AssertFalse(Condition := resultOK, Message := 'Expected PermIntlk NOT OK with local fallback configuration having one FALSE condition');

TEST_FINISHED();
END_METHOD

METHOD PRIVATE GivenNoConfiguration_ExpectDefaultTrueBehavior
VAR
    resultOK : BOOL;
END_VAR
TEST(__POUNAME());

// Initialize without injecting any configuration (pure default behavior)
TestPermIntlk[9].Initialize();

// Don't configure anything - no injection, no local configuration changes
// This should result in default TRUE behavior as per user requirement

// Run cyclic evaluation
TestPermIntlk[9].CyclicLogic();

// Check result - should be TRUE when no configuration is provided
resultOK := TestPermIntlk[9].P_OK;

AssertTrue(Condition := resultOK, Message := 'Expected PermIntlk OK when no configuration is provided (default TRUE behavior)');

TEST_FINISHED();
END_METHOD

METHOD PRIVATE GivenOneConditionFalse_WhenModeAllConditions_ExpectPermIntlkNotOK
VAR
    resultOK : BOOL;
END_VAR
TEST(__POUNAME());

// Initialize the PermIntlk
TestPermIntlk[1].Initialize();

// Configure for "All Conditions Must Be Met" mode
TestPermIntlk[1].P_PermIntlkConfiguration.Mode := E_ModePermIntlk.IfAllConditionsMet;

// Set up test conditions - one FALSE
TestPermIntlk[1].P_PermIntlkConfiguration.PermIntlkObj[0].Description := 'Test Condition 1 - OK';
TestPermIntlk[1].P_PermIntlkConfiguration.PermIntlkObj[0].Condition := TRUE;
TestPermIntlk[1].P_PermIntlkConfiguration.PermIntlkObj[1].Description := 'Test Condition 2 - FAIL';
TestPermIntlk[1].P_PermIntlkConfiguration.PermIntlkObj[1].Condition := FALSE;
TestPermIntlk[1].P_PermIntlkConfiguration.PermIntlkObj[2].Description := 'Test Condition 3 - OK';
TestPermIntlk[1].P_PermIntlkConfiguration.PermIntlkObj[2].Condition := TRUE;

// Run cyclic evaluation
TestPermIntlk[1].CyclicLogic();

// Check result
resultOK := TestPermIntlk[1].P_OK;

AssertFalse(Condition := resultOK, Message := 'Expected PermIntlk NOT OK when one condition is FALSE in AllConditions mode');

TEST_FINISHED();
END_METHOD

METHOD PRIVATE GivenOneConditionTrue_WhenModeAnyConditions_ExpectPermIntlkOK
VAR
    resultOK : BOOL;
END_VAR
TEST(__POUNAME());

// Initialize the PermIntlk
TestPermIntlk[4].Initialize();

// Configure for "Any Condition Met" mode
TestPermIntlk[4].P_PermIntlkConfiguration.Mode := E_ModePermIntlk.IfAnyConditionMet;

// Set up test conditions - one TRUE
TestPermIntlk[4].P_PermIntlkConfiguration.PermIntlkObj[0].Description := 'Test Condition 1 - FAIL';
TestPermIntlk[4].P_PermIntlkConfiguration.PermIntlkObj[0].Condition := FALSE;
TestPermIntlk[4].P_PermIntlkConfiguration.PermIntlkObj[1].Description := 'Test Condition 2 - OK';
TestPermIntlk[4].P_PermIntlkConfiguration.PermIntlkObj[1].Condition := TRUE;
TestPermIntlk[4].P_PermIntlkConfiguration.PermIntlkObj[2].Description := 'Test Condition 3 - FAIL';
TestPermIntlk[4].P_PermIntlkConfiguration.PermIntlkObj[2].Condition := FALSE;

// Run cyclic evaluation
TestPermIntlk[4].CyclicLogic();

// Check result
resultOK := TestPermIntlk[4].P_OK;

AssertTrue(Condition := resultOK, Message := 'Expected PermIntlk OK when one condition is TRUE in AnyCondition mode');

TEST_FINISHED();
END_METHOD

METHOD PRIVATE GivenUnconfiguredConditions_ExpectDefaultTrueBehavior
VAR
    resultOK : BOOL;
END_VAR
TEST(__POUNAME());

// Initialize the PermIntlk without configuring conditions (default behavior)
TestPermIntlk[6].Initialize();

// Configure for "All Conditions Must Be Met" mode
TestPermIntlk[6].P_PermIntlkConfiguration.Mode := E_ModePermIntlk.IfAllConditionsMet;

// Don't configure any conditions - they should default to TRUE
// Default Description should be 'PermIntlk Condition Not Configured'
// Default Condition should be TRUE

// Run cyclic evaluation
TestPermIntlk[6].CyclicLogic();

// Check result
resultOK := TestPermIntlk[6].P_OK;

AssertTrue(Condition := resultOK, Message := 'Expected PermIntlk OK with unconfigured conditions (default TRUE behavior)');

TEST_FINISHED();
END_METHOD

METHOD PRIVATE TEST_ConfigResolution_RecoversToInjected_WhenRefsValidAgain
VAR
    resolution : E_ConfigurationResolution;
    resultOK : BOOL;
END_VAR
TEST(__POUNAME());

// Start with local configuration (simulate recovery scenario)
TestPermIntlk[41].Initialize();
TestPermIntlk[41].P_PermIntlkConfiguration.Mode := E_ModePermIntlk.IfAllConditionsMet;
TestPermIntlk[41].P_PermIntlkConfiguration.PermIntlkObj[0].Description := 'Local Config';
TestPermIntlk[41].P_PermIntlkConfiguration.PermIntlkObj[0].Condition := TRUE;
TestPermIntlk[41].CyclicLogic();

// Verify using local configuration
resolution := TestPermIntlk[41].PermIntlkStatus.PermIntlkConfigResolution;
AssertEquals_DINT(Expected := TO_DINT(E_ConfigurationResolution.Local), Actual := TO_DINT(resolution), Message := 'Should initially use local configuration');

// Now inject valid configuration (simulate recovery)
TestPermIntlkCmd[41].Initialize();
TestPermIntlkCmd[41].P_PermIntlkConfiguration.Mode := E_ModePermIntlk.IfAllConditionsMet;
TestPermIntlkCmd[41].P_PermIntlkConfiguration.PermIntlkObj[0].Description := 'Recovered Injected';
TestPermIntlkCmd[41].P_PermIntlkConfiguration.PermIntlkObj[0].Condition := TRUE;

iTestPermIntlkConfig := TestPermIntlkCmd[41];
TestPermIntlk[41].InjectPermIntlkConfiguration(iTestPermIntlkConfig);
TestPermIntlk[41].Initialize(); // Re-initialize to trigger resolution check
TestPermIntlk[41].CyclicLogic();

// Verify recovery to injected configuration
resolution := TestPermIntlk[41].PermIntlkStatus.PermIntlkConfigResolution;
resultOK := TestPermIntlk[41].P_OK;

AssertEquals_DINT(Expected := TO_DINT(E_ConfigurationResolution.InjectedInterface), Actual := TO_DINT(resolution), Message := 'Should recover to injected configuration when refs valid again');
AssertTrue(Condition := resultOK, Message := 'Should still function with recovered injected config');

TEST_FINISHED();
END_METHOD

METHOD PRIVATE TEST_ConfigResolution_SwitchesInjectedToLocal_WhenRefsInvalid
VAR
    resolution : E_ConfigurationResolution;
    resultOK : BOOL;
END_VAR
TEST(__POUNAME());

// Set up valid injected configuration initially
TestPermIntlkCmd[40].Initialize();
TestPermIntlkCmd[40].P_PermIntlkConfiguration.Mode := E_ModePermIntlk.IfAllConditionsMet;
TestPermIntlkCmd[40].P_PermIntlkConfiguration.PermIntlkObj[0].Description := 'Valid Injected';
TestPermIntlkCmd[40].P_PermIntlkConfiguration.PermIntlkObj[0].Condition := TRUE;

// Inject and initialize
iTestPermIntlkConfig := TestPermIntlkCmd[40];
TestPermIntlk[40].InjectPermIntlkConfiguration(iTestPermIntlkConfig);
TestPermIntlk[40].Initialize();
TestPermIntlk[40].CyclicLogic();

// Verify initially using injected configuration
resolution := TestPermIntlk[40].PermIntlkStatus.PermIntlkConfigResolution;
AssertEquals_DINT(Expected := TO_DINT(E_ConfigurationResolution.InjectedInterface), Actual := TO_DINT(resolution), Message := 'Should initially use injected configuration');

// Simulate invalid references by injecting null/invalid configuration
// This would normally happen if the injected interface becomes invalid
TestPermIntlk[40].InjectPermIntlkConfiguration(iPermIntlkCfg := 0);
TestPermIntlk[40].Initialize(); // Re-initialize to trigger resolution check

// Configure local fallback
TestPermIntlk[40].P_PermIntlkConfiguration.Mode := E_ModePermIntlk.IfAllConditionsMet;
TestPermIntlk[40].P_PermIntlkConfiguration.PermIntlkObj[0].Description := 'Local Fallback';
TestPermIntlk[40].P_PermIntlkConfiguration.PermIntlkObj[0].Condition := TRUE;

TestPermIntlk[40].CyclicLogic();

// Verify switch to local configuration
resolution := TestPermIntlk[40].PermIntlkStatus.PermIntlkConfigResolution;
resultOK := TestPermIntlk[40].P_OK;

AssertEquals_DINT(Expected := TO_DINT(E_ConfigurationResolution.Local), Actual := TO_DINT(resolution), Message := 'Should switch to local configuration when injected refs invalid');
AssertTrue(Condition := resultOK, Message := 'Should still function with local fallback');

TEST_FINISHED();
END_METHOD

METHOD PRIVATE TEST_ConfiguredFlag_EmptyDescription_TreatedAsUnconfigured
VAR
    configuredFlag1, configuredFlag2, configuredFlag3 : BOOL;
    resultOK : BOOL;
END_VAR
TEST(__POUNAME());

// Initialize and configure conditions with various description states
TestPermIntlk[50].Initialize();
TestPermIntlk[50].P_PermIntlkConfiguration.Mode := E_ModePermIntlk.IfAllConditionsMet;

// Condition 0: Empty description (should be unconfigured)
TestPermIntlk[50].P_PermIntlkConfiguration.PermIntlkObj[0].Description := '';
TestPermIntlk[50].P_PermIntlkConfiguration.PermIntlkObj[0].Condition := FALSE;

// Condition 1: Default "not configured" description (should be unconfigured)
TestPermIntlk[50].P_PermIntlkConfiguration.PermIntlkObj[1].Description := 'PermIntlk Condition Not Configured';
TestPermIntlk[50].P_PermIntlkConfiguration.PermIntlkObj[1].Condition := FALSE;

// Condition 2: Actual description (should be configured)
TestPermIntlk[50].P_PermIntlkConfiguration.PermIntlkObj[2].Description := 'Valid Configuration';
TestPermIntlk[50].P_PermIntlkConfiguration.PermIntlkObj[2].Condition := TRUE;

// Run evaluation to trigger configuration analysis
TestPermIntlk[50].CyclicLogic();

// Check configured flags
configuredFlag1 := TestPermIntlk[50].PermIntlkStatus.ConditionStatus[0].Configured;
configuredFlag2 := TestPermIntlk[50].PermIntlkStatus.ConditionStatus[1].Configured;
configuredFlag3 := TestPermIntlk[50].PermIntlkStatus.ConditionStatus[2].Configured;
resultOK := TestPermIntlk[50].P_OK;

AssertFalse(Condition := configuredFlag1, Message := 'Empty description should be treated as unconfigured');
AssertFalse(Condition := configuredFlag2, Message := 'Default description should be treated as unconfigured');
AssertTrue(Condition := configuredFlag3, Message := 'Valid description should be treated as configured');

// Since only one condition is configured and it's TRUE, result should be TRUE
// (unconfigured conditions default to safe state)
AssertTrue(Condition := resultOK, Message := 'P_OK should be TRUE when only configured condition is TRUE');

TEST_FINISHED();
END_METHOD

METHOD PRIVATE TEST_Initialize_Twice_IsIdempotent_NoDuplicateSideEffects
VAR
    resultOK1, resultOK2 : BOOL;
    resolution1, resolution2 : E_ConfigurationResolution;
END_VAR
TEST(__POUNAME());

// Set up configuration
TestPermIntlkCmd[20].Initialize();
TestPermIntlkCmd[20].P_PermIntlkConfiguration.Mode := E_ModePermIntlk.IfAllConditionsMet;
TestPermIntlkCmd[20].P_PermIntlkConfiguration.PermIntlkObj[0].Description := 'Idempotent Test';
TestPermIntlkCmd[20].P_PermIntlkConfiguration.PermIntlkObj[0].Condition := TRUE;

// Inject and initialize first time
iTestPermIntlkConfig := TestPermIntlkCmd[20];
TestPermIntlk[20].InjectPermIntlkConfiguration(iTestPermIntlkConfig);
TestPermIntlk[20].Initialize();
TestPermIntlk[20].CyclicLogic();

// Capture first state
resultOK1 := TestPermIntlk[20].P_OK;
resolution1 := TestPermIntlk[20].PermIntlkStatus.PermIntlkConfigResolution;

// Initialize second time (should be idempotent)
TestPermIntlk[20].Initialize();
TestPermIntlk[20].CyclicLogic();

// Capture second state
resultOK2 := TestPermIntlk[20].P_OK;
resolution2 := TestPermIntlk[20].PermIntlkStatus.PermIntlkConfigResolution;

// Results should be identical
AssertEquals_BOOL(Expected := resultOK1, Actual := resultOK2, Message := 'P_OK should be identical after second initialization');
AssertEquals_DINT(Expected := TO_DINT(resolution1), Actual := TO_DINT(resolution2), Message := 'Resolution should be identical after second initialization');

TEST_FINISHED();
END_METHOD

METHOD PRIVATE TEST_Permissive_Fall_LogsInterlockLost_Once
VAR
    resultOK : BOOL;
END_VAR
TEST(__POUNAME());

// Set up configuration with condition initially TRUE
TestPermIntlkCmd[11].Initialize();
TestPermIntlkCmd[11].P_PermIntlkConfiguration.Mode := E_ModePermIntlk.IfAllConditionsMet;
TestPermIntlkCmd[11].P_PermIntlkConfiguration.PermIntlkObj[0].Description := 'Test Condition Fall';
TestPermIntlkCmd[11].P_PermIntlkConfiguration.PermIntlkObj[0].Condition := TRUE;

// Inject and initialize
iTestPermIntlkConfig := TestPermIntlkCmd[11];
TestPermIntlk[11].InjectPermIntlkConfiguration(iTestPermIntlkConfig);
TestPermIntlk[11].Initialize();

// First cycle - should be TRUE
TestPermIntlk[11].CyclicLogic();
resultOK := TestPermIntlk[11].P_OK;
AssertTrue(Condition := resultOK, Message := 'Initial state should be TRUE');

// Change condition to FALSE - this should trigger falling edge log
TestPermIntlkCmd[11].P_PermIntlkConfiguration.PermIntlkObj[0].Condition := FALSE;
TestPermIntlk[11].CyclicLogic();
resultOK := TestPermIntlk[11].P_OK;
AssertFalse(Condition := resultOK, Message := 'After fall, P_OK should be FALSE');

// Additional cycles should not retrigger log (no log spam)
TestPermIntlk[11].CyclicLogic();
TestPermIntlk[11].CyclicLogic();
resultOK := TestPermIntlk[11].P_OK;
AssertFalse(Condition := resultOK, Message := 'P_OK should remain FALSE on subsequent cycles');

TEST_FINISHED();
END_METHOD

METHOD PRIVATE TEST_Permissive_Rise_LogsPermissiveOK_Once
VAR
    resultOK : BOOL;
END_VAR
TEST(__POUNAME());

// Set up configuration with condition initially FALSE
TestPermIntlkCmd[10].Initialize();
TestPermIntlkCmd[10].P_PermIntlkConfiguration.Mode := E_ModePermIntlk.IfAllConditionsMet;
TestPermIntlkCmd[10].P_PermIntlkConfiguration.PermIntlkObj[0].Description := 'Test Condition Rise';
TestPermIntlkCmd[10].P_PermIntlkConfiguration.PermIntlkObj[0].Condition := FALSE;

// Inject and initialize
iTestPermIntlkConfig := TestPermIntlkCmd[10];
TestPermIntlk[10].InjectPermIntlkConfiguration(iTestPermIntlkConfig);
TestPermIntlk[10].Initialize();

// First cycle - should be FALSE, no logs yet
TestPermIntlk[10].CyclicLogic();
resultOK := TestPermIntlk[10].P_OK;
AssertFalse(Condition := resultOK, Message := 'Initial state should be FALSE');

// Change condition to TRUE - this should trigger rising edge log
TestPermIntlkCmd[10].P_PermIntlkConfiguration.PermIntlkObj[0].Condition := TRUE;
TestPermIntlk[10].CyclicLogic();
resultOK := TestPermIntlk[10].P_OK;
AssertTrue(Condition := resultOK, Message := 'After rise, P_OK should be TRUE');

// Additional cycles should not retrigger log (no log spam)
TestPermIntlk[10].CyclicLogic();
TestPermIntlk[10].CyclicLogic();
resultOK := TestPermIntlk[10].P_OK;
AssertTrue(Condition := resultOK, Message := 'P_OK should remain TRUE on subsequent cycles');

TEST_FINISHED();
END_METHOD

METHOD PRIVATE TEST_Permissive_Toggle_NoLogSpam
VAR
    resultOK : BOOL;
    toggleCount : DINT;
END_VAR
TEST(__POUNAME());

// Set up configuration with condition initially FALSE
TestPermIntlkCmd[12].Initialize();
TestPermIntlkCmd[12].P_PermIntlkConfiguration.Mode := E_ModePermIntlk.IfAllConditionsMet;
TestPermIntlkCmd[12].P_PermIntlkConfiguration.PermIntlkObj[0].Description := 'Test Condition Toggle';
TestPermIntlkCmd[12].P_PermIntlkConfiguration.PermIntlkObj[0].Condition := FALSE;

// Inject and initialize
iTestPermIntlkConfig := TestPermIntlkCmd[12];
TestPermIntlk[12].InjectPermIntlkConfiguration(iTestPermIntlkConfig);
TestPermIntlk[12].Initialize();

// Initial cycle
TestPermIntlk[12].CyclicLogic();

// Toggle multiple times to verify edge-triggered behavior
FOR toggleCount := 1 TO 5 BY 1 DO
    // FALSE -> TRUE (rising edge)
    TestPermIntlkCmd[12].P_PermIntlkConfiguration.PermIntlkObj[0].Condition := TRUE;
    TestPermIntlk[12].CyclicLogic();
    resultOK := TestPermIntlk[12].P_OK;
    AssertTrue(Condition := resultOK, Message := 'Should be TRUE after rising edge');

    // Stay TRUE for a cycle (no additional logs)
    TestPermIntlk[12].CyclicLogic();

    // TRUE -> FALSE (falling edge)
    TestPermIntlkCmd[12].P_PermIntlkConfiguration.PermIntlkObj[0].Condition := FALSE;
    TestPermIntlk[12].CyclicLogic();
    resultOK := TestPermIntlk[12].P_OK;
    AssertFalse(Condition := resultOK, Message := 'Should be FALSE after falling edge');

    // Stay FALSE for a cycle (no additional logs)
    TestPermIntlk[12].CyclicLogic();
END_FOR

TEST_FINISHED();
END_METHOD

METHOD PRIVATE TEST_ReinitObjects_ClearsLocalConfig_AndSetsP_OK_TRUE
VAR
    resultOK : BOOL;
    conditionDescription : STRING;
END_VAR
TEST(__POUNAME());

// Initialize and configure local configuration
TestPermIntlk[21].Initialize();
TestPermIntlk[21].P_PermIntlkConfiguration.Mode := E_ModePermIntlk.IfAllConditionsMet;
TestPermIntlk[21].P_PermIntlkConfiguration.PermIntlkObj[0].Description := 'Before Reinit';
TestPermIntlk[21].P_PermIntlkConfiguration.PermIntlkObj[0].Condition := FALSE;

// Run logic to get into known state
TestPermIntlk[21].CyclicLogic();
resultOK := TestPermIntlk[21].P_OK;
AssertFalse(Condition := resultOK, Message := 'Should be FALSE before reinit');

// Call ReinitObjects
TestPermIntlk[21].ReinitObjects();

// Verify local config is cleared and P_OK is TRUE
resultOK := TestPermIntlk[21].P_OK;
conditionDescription := TestPermIntlk[21].P_PermIntlkConfiguration.PermIntlkObj[0].Description;

AssertTrue(Condition := resultOK, Message := 'P_OK should be TRUE after ReinitObjects');
AssertEquals_STRING(Expected := 'PermIntlk Condition Not Configured', Actual := conditionDescription, Message := 'Description should be cleared after ReinitObjects');

TEST_FINISHED();
END_METHOD

METHOD PRIVATE TEST_RuntimeConfigLoss_InjectedRefsInvalidatedDuringExecution
VAR
    resolution : E_ConfigurationResolution;
    resultOK : BOOL;
    conditionDescription : STRING;
END_VAR
TEST(__POUNAME());

// Purpose: Test actual runtime configuration loss scenario where injected references
// become invalid during execution without explicit re-injection
// This validates our _EvaluateConfiguration fix that detects resolution changes

// === STEP 1: Set up valid injected configuration ===
TestPermIntlkCmd[60].Initialize();
TestPermIntlkCmd[60].P_PermIntlkConfiguration.Mode := E_ModePermIntlk.IfAllConditionsMet;
TestPermIntlkCmd[60].P_PermIntlkConfiguration.PermIntlkObj[0].Description := 'Runtime Valid Config';
TestPermIntlkCmd[60].P_PermIntlkConfiguration.PermIntlkObj[0].Condition := TRUE;

// Inject and initialize normally
iTestPermIntlkConfig := TestPermIntlkCmd[60];
TestPermIntlk[60].InjectPermIntlkConfiguration(iTestPermIntlkConfig);
TestPermIntlk[60].Initialize();
TestPermIntlk[60].CyclicLogic();

// Verify initially using injected configuration
resolution := TestPermIntlk[60].PermIntlkStatus.PermIntlkConfigResolution;
resultOK := TestPermIntlk[60].P_OK;
AssertEquals_DINT(Expected := TO_DINT(E_ConfigurationResolution.InjectedInterface), Actual := TO_DINT(resolution), Message := 'Should initially use injected configuration');
AssertTrue(Condition := resultOK, Message := 'Should be OK with valid injected configuration');

// === STEP 2: Set up local fallback configuration ===
// Configure distinctive local configuration for fallback
TestPermIntlk[60].P_PermIntlkConfiguration.Mode := E_ModePermIntlk.IfAllConditionsMet;
TestPermIntlk[60].P_PermIntlkConfiguration.PermIntlkObj[0].Description := 'Runtime Local Fallback';
TestPermIntlk[60].P_PermIntlkConfiguration.PermIntlkObj[0].Condition := TRUE;

// === STEP 3: Simulate runtime reference invalidation ===
// This simulates what happens when network connections are lost, memory corruption occurs,
// or external systems become unavailable - WITHOUT calling InjectPermIntlkConfiguration again
// We simulate this by calling InjectPermIntlkConfiguration with null to trigger the runtime scenario
TestPermIntlk[60].InjectPermIntlkConfiguration(iPermIntlkCfg := 0);  // Simulate reference becoming invalid

// === STEP 4: Trigger resolution change detection through CyclicLogic ===
// Our fix should detect the resolution change and update references
TestPermIntlk[60].CyclicLogic();

// === STEP 5: Verify automatic fallback to local configuration ===
resolution := TestPermIntlk[60].PermIntlkStatus.PermIntlkConfigResolution;
resultOK := TestPermIntlk[60].P_OK;
conditionDescription := TestPermIntlk[60].P_PermIntlkConfiguration.PermIntlkObj[0].Description;

AssertEquals_DINT(Expected := TO_DINT(E_ConfigurationResolution.Local), Actual := TO_DINT(resolution), Message := 'RUNTIME FIX: Should automatically switch to local configuration when injected refs become invalid');
AssertTrue(Condition := resultOK, Message := 'Should continue functioning with local fallback configuration');
AssertEquals_STRING(Expected := 'Runtime Local Fallback', Actual := conditionDescription, Message := 'Should use local fallback configuration description');

// === STEP 6: Verify continued operation ===
// Run multiple cycles to ensure stable operation with local configuration
TestPermIntlk[60].CyclicLogic();
TestPermIntlk[60].CyclicLogic();
TestPermIntlk[60].CyclicLogic();

resolution := TestPermIntlk[60].PermIntlkStatus.PermIntlkConfigResolution;
resultOK := TestPermIntlk[60].P_OK;

AssertEquals_DINT(Expected := TO_DINT(E_ConfigurationResolution.Local), Actual := TO_DINT(resolution), Message := 'Should maintain local configuration resolution consistently');
AssertTrue(Condition := resultOK, Message := 'Should maintain stable operation with local configuration');

TEST_FINISHED();
END_METHOD

METHOD PRIVATE TEST_RuntimeConfigRecovery_ValidRefsRestoredDuringExecution
VAR
    resolution : E_ConfigurationResolution;
    resultOK : BOOL;
    conditionDescription : STRING;
END_VAR
TEST(__POUNAME());

// Purpose: Test runtime configuration recovery scenario where injected references
// are restored during execution after being invalid
// This validates our _EvaluateConfiguration fix for bidirectional resolution changes

// === STEP 1: Start with local configuration ===
TestPermIntlk[61].Initialize();
TestPermIntlk[61].P_PermIntlkConfiguration.Mode := E_ModePermIntlk.IfAllConditionsMet;
TestPermIntlk[61].P_PermIntlkConfiguration.PermIntlkObj[0].Description := 'Recovery Local Config';
TestPermIntlk[61].P_PermIntlkConfiguration.PermIntlkObj[0].Condition := TRUE;
TestPermIntlk[61].CyclicLogic();

// Verify starting with local configuration
resolution := TestPermIntlk[61].PermIntlkStatus.PermIntlkConfigResolution;
AssertEquals_DINT(Expected := TO_DINT(E_ConfigurationResolution.Local), Actual := TO_DINT(resolution), Message := 'Should start with local configuration');

// === STEP 2: Set up distinctive injected configuration ===
TestPermIntlkCmd[61].Initialize();
TestPermIntlkCmd[61].P_PermIntlkConfiguration.Mode := E_ModePermIntlk.IfAllConditionsMet;
TestPermIntlkCmd[61].P_PermIntlkConfiguration.PermIntlkObj[0].Description := 'Recovery Injected Config';
TestPermIntlkCmd[61].P_PermIntlkConfiguration.PermIntlkObj[0].Condition := TRUE;

// === STEP 3: Simulate runtime reference restoration ===
// This simulates what happens when network connections are restored, external systems
// come back online, or memory references are re-established - WITHOUT calling Initialize again
// We restore the interface reference to simulate runtime recovery
iTestPermIntlkConfig := TestPermIntlkCmd[61];
TestPermIntlk[61].InjectPermIntlkConfiguration(iTestPermIntlkConfig);  // Simulate reference becoming valid again

// === STEP 4: Trigger resolution change detection through CyclicLogic ===
// Our fix should detect the resolution change and update references
TestPermIntlk[61].CyclicLogic();

// === STEP 5: Verify automatic recovery to injected configuration ===
resolution := TestPermIntlk[61].PermIntlkStatus.PermIntlkConfigResolution;
resultOK := TestPermIntlk[61].P_OK;

AssertEquals_DINT(Expected := TO_DINT(E_ConfigurationResolution.InjectedInterface), Actual := TO_DINT(resolution), Message := 'RUNTIME FIX: Should automatically switch to injected configuration when refs become valid');
AssertTrue(Condition := resultOK, Message := 'Should function correctly with recovered injected configuration');

// === STEP 6: Verify recovered configuration is being used ===
// Access the configuration through the public property to verify it's the injected one
conditionDescription := TestPermIntlk[61].P_PermIntlkConfiguration.PermIntlkObj[0].Description;
AssertEquals_STRING(Expected := 'Recovery Injected Config', Actual := conditionDescription, Message := 'Should use recovered injected configuration description');

// === STEP 7: Verify continued stable operation ===
// Run multiple cycles to ensure stable operation with recovered configuration
TestPermIntlk[61].CyclicLogic();
TestPermIntlk[61].CyclicLogic();
TestPermIntlk[61].CyclicLogic();

resolution := TestPermIntlk[61].PermIntlkStatus.PermIntlkConfigResolution;
resultOK := TestPermIntlk[61].P_OK;

AssertEquals_DINT(Expected := TO_DINT(E_ConfigurationResolution.InjectedInterface), Actual := TO_DINT(resolution), Message := 'Should maintain injected configuration resolution consistently');
AssertTrue(Condition := resultOK, Message := 'Should maintain stable operation with recovered configuration');

TEST_FINISHED();
END_METHOD

METHOD PRIVATE TEST_SetElementIndices_AssignsMissingIndices_ForInjectedConfig
VAR
    index0, index1, index2 : DINT;
END_VAR
TEST(__POUNAME());

// Set up configuration with indices set to 0 (uninitialized)
TestPermIntlkCmd[30].Initialize();
TestPermIntlkCmd[30].P_PermIntlkConfiguration.PermIntlkObj[0].Description := 'Auto-Index Test 0';
TestPermIntlkCmd[30].P_PermIntlkConfiguration.PermIntlkObj[0].Index := 0; // Should be auto-assigned
TestPermIntlkCmd[30].P_PermIntlkConfiguration.PermIntlkObj[1].Description := 'Auto-Index Test 1';
TestPermIntlkCmd[30].P_PermIntlkConfiguration.PermIntlkObj[1].Index := 0; // Should be auto-assigned
TestPermIntlkCmd[30].P_PermIntlkConfiguration.PermIntlkObj[2].Description := 'Auto-Index Test 2';
TestPermIntlkCmd[30].P_PermIntlkConfiguration.PermIntlkObj[2].Index := 0; // Should be auto-assigned

// Inject and initialize (this should trigger _SetElementIndices)
iTestPermIntlkConfig := TestPermIntlkCmd[30];
TestPermIntlk[30].InjectPermIntlkConfiguration(iTestPermIntlkConfig);
TestPermIntlk[30].Initialize();

// Check that indices have been auto-assigned
index0 := TestPermIntlkCmd[30].P_PermIntlkConfiguration.PermIntlkObj[0].Index;
index1 := TestPermIntlkCmd[30].P_PermIntlkConfiguration.PermIntlkObj[1].Index;
index2 := TestPermIntlkCmd[30].P_PermIntlkConfiguration.PermIntlkObj[2].Index;

AssertEquals_DINT(Expected := 0, Actual := index0, Message := 'Index 0 should be auto-assigned');
AssertEquals_DINT(Expected := 1, Actual := index1, Message := 'Index 1 should be auto-assigned');
AssertEquals_DINT(Expected := 2, Actual := index2, Message := 'Index 2 should be auto-assigned');

TEST_FINISHED();
END_METHOD

END_FUNCTION_BLOCK

// Tests/FB_CommandTestsI
FUNCTION_BLOCK FB_CommandTestsI EXTENDS TcUnit.FB_TestSuite
VAR CONSTANT
	// Test method index constants - one unique index per test method (0-113)

	// GivenCommand* helper test methods (0-25)
	INDEX_GIVENCOMMAND_WHENCANCEL_EXPECTREMOVEDFROMQUEUE							: DINT := 0;
	INDEX_GIVENCOMMAND_WHENCYCLICLOGICCALLED_EXPECTUPDATED							: DINT := 1;
	INDEX_GIVENCOMMAND_WHENEXECUTECALLED_EXPECTEXECUTION							: DINT := 2;
	INDEX_GIVENCOMMAND_WHENPAUSECALLED_EXPECTCOMMANDPAUSES							: DINT := 3;
	INDEX_GIVENCOMMAND_WHENQUEUECALLED_EXPECTADDEDTOQUEUE							: DINT := 4;
	INDEX_GIVENCOMMAND_WHENRESETCALLED_EXPECTSTATECLEARED							: DINT := 5;
	INDEX_GIVENCOMMAND_WHENRESUMECALLED_EXPECTCOMMANDRESUMES						: DINT := 6;
	INDEX_GIVENCOMMAND_WHENVALIDATECALLED_EXPECTPERMISSIVEOK						: DINT := 7;
	INDEX_GIVENCOMMAND_WHENVALIDATECALLED_EXPECTMATCHCONFIG							: DINT := 8;
	INDEX_GIVENCOMMANDALREADYRUNNING_WHENEXECUTE_CONFLICT							: DINT := 9;
	INDEX_GIVENCOMMANDEXECUTED_WHENCYCLICLOGICRUNS_EXPECTSTATEPROGRESSION			: DINT := 10;
	INDEX_GIVENCOMMANDINIDLESTATE_WHENCANCEL_EXPECTNOACTIONTAKEN					: DINT := 11;
	INDEX_GIVENCOMMANDINVALID_WHENVALIDATECALLED_EXPECTFALSE						: DINT := 12;
	INDEX_GIVENCOMMANDPAUSED_WHENABORT_EXPECTCOMMANDABORTEDANDSTATUSUPDATED			: DINT := 13;
	INDEX_GIVENCOMMANDPAUSED_WHENRESUME_EXPECTCOMMANDRESUMESEXECUTION				: DINT := 14;
	INDEX_GIVENCOMMANDQUEUED_WHENABORT_EXPECTCOMMANDABORTEDANDSTATUSUPDATED			: DINT := 15;
	INDEX_GIVENCOMMANDQUEUED_WHENCANCEL_EXPECTCOMMANDREMOVEDFROMQUEUE				: DINT := 16;
	INDEX_GIVENCOMMANDVALIDATED_WHENVALIDATECALLED_EXPECTTRUE						: DINT := 17;
	INDEX_GIVENCOMPONENTRESET_WHENRESETCALLED_EXPECTALLCOMMANDSTATECLEARED			: DINT := 18;
	INDEX_GIVENINJECTEDCONFIGURATIONSVALID_EXPECTINTERFACESSTOREDANDINITIALIZED		: DINT := 19;
	INDEX_GIVENINVALIDCONFIGURATION_WHENINJECTCONFIGURATIONCALLED_EXPECTINITFAILURE	: DINT := 20;
	INDEX_GIVENINVALIDCONFIGURATIONS_WHENINJECTCONFIGURATIONS_EXPECTINITFAILURE		: DINT := 21;
	INDEX_GIVENRUNNINGCOMMAND_WHENPAUSE_EXPECTCOMMANDTRANSITIONSTOPAUSEDSTATE		: DINT := 22;
	INDEX_GIVENTIMERSTARTED_WHENCYCLICLOGICRUNS_EXPECTELAPSEDTIMEINCREASES			: DINT := 23;
	INDEX_GIVENTIMERSTOPPED_WHENCYCLICLOGICRUNS_EXPECTELAPSEDTIMEREMAINCONSTANT		: DINT := 24;
	INDEX_GIVENVALIDCONFIGURATION_WHENINJECTCONFIGURATIONCALLED_EXPECTCONFIGSTORED	: DINT := 25;

	// TEST_* methods (26-113)
	INDEX_ABORT_AFTERCOMPLETE_IGNOREDWITHWARNING									: DINT := 26;
	INDEX_ABORT_ERRORCLASSIFICATION													: DINT := 27;
	INDEX_ABORT_WHENIDLEQUEUED_SETSRESULTABORTED									: DINT := 28;
	INDEX_ABORTAFTERCOMPLETE_STATEPRESERVATION										: DINT := 29;
	INDEX_ABORTDURINGCOMPLETIONWAIT													: DINT := 30;
	INDEX_ACCEPTEDCOMMAND_WHENEXECUTED_RESULTBECOMESOK								: DINT := 31;
	INDEX_BADREQUEST_INTERLOCKMISCONFIGURED											: DINT := 32;
	INDEX_BUSYCOMMANDELAPSEDTIMEEQUALS_COMMANDABORTED								: DINT := 33;
	INDEX_CANCEL_FROMQUEUEDSTATE													: DINT := 34;
	INDEX_CANCEL_REMOVESCOMMANDFROMQUEUE											: DINT := 35;
	INDEX_CANCEL_SETSCOMMANDSTATUSTOCANCELLED										: DINT := 36;
	INDEX_CANCEL_SETSRESULTCANCELLED												: DINT := 37;
	INDEX_CANCEL_WHENBUSY_REJECTED_NOCHANGETOSTATE									: DINT := 38;
	INDEX_COMMAND_LOCALREFERENCES_INITIALIZEDPROPERLY								: DINT := 39;
	INDEX_COMMAND_MISSINGCONFIGINTERFACE_FALLBACK									: DINT := 40;
	INDEX_COMMAND_PERMINTLKCHILD_INITIALIZED										: DINT := 41;
	INDEX_COMMANDATTEMPTSEXCEEDRETRYCOUNT											: DINT := 42;
	INDEX_COMMANDCOMPLETES_STATUSDONEANDCLEARED										: DINT := 43;
	INDEX_COMMANDSTATUS_CONFIGREF_POINTSTOCONFIGURATION								: DINT := 44;
	INDEX_COMMANDTIMEOUT_TRIGGERSRESET												: DINT := 45;
	INDEX_COMPLETE_ERROR_PERSISTSUNTILRESET											: DINT := 46;
	INDEX_COMPLETE_OK_AUTORESETNEXTCYCLE											: DINT := 47;
	INDEX_COMPLETESTATE_PRESERVESABORTEDRESULT										: DINT := 48;
	INDEX_COMPLETESTATE_PRESERVESTIMEOUTRESULT										: DINT := 49;
	INDEX_COMPLETESTATE_SETSOKFORSUCCESSFUL											: DINT := 50;
	INDEX_COMPLETIONCALLBACKTOSEQUENCER												: DINT := 51;
	INDEX_COMPLETIONCONDITIONEVALUATION												: DINT := 52;
	INDEX_COMPLETIONCONDITIONWITHTIMEOUT											: DINT := 53;
	INDEX_COMPLETIONWITHINTERLOCKDROP												: DINT := 54;
	INDEX_COMPLEXCOMPLETIONCONDITION												: DINT := 55;
	INDEX_COMPONENTBUSY_DURINGVALIDATION_RESULTCONFLICT								: DINT := 56;
	INDEX_CONFIG_FALLBACKTOLOCAL_WHENINJECTEDINVALID								: DINT := 57;
	INDEX_CONFIG_RECOVERYTOINJECTED_WHENVALIDAGAIN									: DINT := 58;
	INDEX_CONFIGURATIONRESOLUTION_HANDLESVALIDINVALID								: DINT := 59;
	INDEX_CYCLICLOGIC_STATEMACHINEPROGRESSION										: DINT := 60;
	INDEX_DISCRETECOMPLETIONCONDITION												: DINT := 61;
	INDEX_DYNAMICCOMPLETIONCONDITIONUPDATE											: DINT := 62;
	INDEX_EDGETRIGGERED_STATEMACHINEEXECUTION										: DINT := 63;
	INDEX_EXECUTE_HAPPYPATH_TRANSITIONSTOMONITOR									: DINT := 64;
	INDEX_EXECUTE_STATEMACHINEPROGRESSION											: DINT := 65;
	INDEX_EXECUTE_TRANSITIONSFROMACCEPTEDTOOK										: DINT := 66;
	INDEX_EXECUTE_VALIDATESBEFOREACCEPTING											: DINT := 67;
	INDEX_EXECUTE_WHENPERMISSIVEMISSING_RETURNSFORBIDDEN							: DINT := 68;
	INDEX_FASTCOMPLETIONINONESCAN													: DINT := 69;
	INDEX_FORBIDDEN_RESUMEWITHOUTPERMISSIVE											: DINT := 70;
	INDEX_INJECTCONFIGURATIONS_STORESINTERFACES										: DINT := 71;
	INDEX_INTERFACEINJECTIONCONFIGURATIONRESOLUTION									: DINT := 72;
	INDEX_INTERLOCKDROP_ABORTSCOMMANDWHENCONFIGURED									: DINT := 73;
	INDEX_INTERLOCKDROP_FROMMONITORSTATE											: DINT := 74;
	INDEX_INTERLOCKINVALIDCONFIG_DURINGVALIDATION									: DINT := 75;
	INDEX_INTERLOCKLOST_COMPREHENSIVESTATETRANSITIONS								: DINT := 76;
	INDEX_INTERLOCKLOST_FROMEXECUTESTATE											: DINT := 77;
	INDEX_INTERLOCKLOST_SETSCORRECTRESULT											: DINT := 78;
	INDEX_INTERLOCKREFERENCELOST_DURINGEXECUTION									: DINT := 79;
	INDEX_METHODENABLEMENT_BUSYSTATE_ALLOWABORT										: DINT := 80;
	INDEX_METHODENABLEMENT_DONESTATE_ALLOWRESET										: DINT := 81;
	INDEX_METHODENABLEMENT_IDLEWITHINTERLOK_ALLOWEXECUTE							: DINT := 82;
	INDEX_METHODENABLEMENT_IDLEWITHOUTINTERLOK_REJECT								: DINT := 83;
	INDEX_MOTIONCOMPLETIONCONDITION													: DINT := 84;
	INDEX_OPERATIONTOCOMMANDTRANSLATION												: DINT := 85;
	INDEX_OPERATORABORT_VSINTERLOCKABORT_DIFFERENTRESULTS							: DINT := 86;
	INDEX_PAUSERESUME_STATETRANSITIONS												: DINT := 87;
	INDEX_PAUSERESUMEWITHCOMPLETIONCONDITION										: DINT := 88;
	INDEX_PERMINTLKLOST_DURINGBUSY_COMMANDABORTED									: DINT := 89;
	INDEX_PERMISSIVEFALSE_DURINGVALIDATION_FORBIDDEN								: DINT := 90;
	INDEX_QUEUEOPERATIONS_MULTIPLECOMMANDSATOMICITY									: DINT := 91;
	INDEX_RECIPEMANAGERPROVIDESCOMMANDCONFIG										: DINT := 92;
	INDEX_RESET_CLEARSCOMMANDSTATE													: DINT := 93;
	INDEX_RESULTPERSISTENCE_TERMINALSTATES											: DINT := 94;
	INDEX_RETRYCOUNT_INCREMENTONEXECUTIONSTARTONLY									: DINT := 95;
	INDEX_RUNTIMECOMMANDCONFIGLOSS_INJECTEDREFSINVALIDATED							: DINT := 96;
	INDEX_RUNTIMECOMMANDCONFIGRECOVERY_VALIDREFSRESTORED							: DINT := 97;
	INDEX_SLOWCOMPLETIONMULTIPLESCANS												: DINT := 98;
	INDEX_STEPSTATE_TRANSITIONSANDVALIDATION										: DINT := 99;
	INDEX_SYSTEMATICSTATEVALIDATION_IDLESTATES										: DINT := 100;
	INDEX_SYSTEMATICSTATEVALIDATION_TERMINALSTATES									: DINT := 101;
	INDEX_TERMINALRESULTS_ERRORFLAGCONSISTENCY										: DINT := 102;
	INDEX_TIMEBASEDCOMPLETIONCONDITION												: DINT := 103;
	INDEX_TIMEOUTANDINTERLOCKLOST_SAMECYCLE_PRIORITIZE								: DINT := 104;
	INDEX_TIMERCOMPLETIONTIME_SETONCOMMANDCOMPLETE									: DINT := 105;
	INDEX_TIMERINTEGRATION_WITHCOMMANDSTATEMACHINE									: DINT := 106;
	INDEX_TIMERPAUSERESUME_ELAPSEDTIMEACCURACY										: DINT := 107;
	INDEX_TIMERSTOPSONCOMMANDCOMPLETE_NOTTIMEOUT									: DINT := 108;
	INDEX_TIMERTRIGGERTIME_SETONCOMMANDSTART										: DINT := 109;
	INDEX_VALIDATE_RETURNSPROPERRESULT												: DINT := 110;
	INDEX_VALIDATE_WITHCONTINUOUSEVALUATION											: DINT := 111;
	INDEX_VALIDATIONOK_INTERLOCKDROP_DURINGEXECUTION								: DINT := 112;
	INDEX_VALIDCOMMAND_EXPECTEXECUTED												: DINT := 113;

	// Additional indices for multi-scenario tests
	INDEX_TERMINALRESULTS_CLEANCANCEL												: DINT := 114;
	INDEX_TERMINALRESULTS_INTERLOCKLOST											: DINT := 115;
	INDEX_TERMINALRESULTS_TIMEOUT													: DINT := 116;
	INDEX_TERMINALRESULTS_COMPLETE_OK												: DINT := 117;
	INDEX_TERMINALRESULTS_COMPLETE_ERROR											: DINT := 118;
	INDEX_VALIDATIONOK_INTERLOCKDROP_SCENARIO2										: DINT := 119;

	// Fixed duplicate indices - these tests were incorrectly reusing other test indices
	INDEX_TIMEOUTANDINTERLOCKLOST_SAMECYCLE_PRIORITIZEINTERLOCKLOST					: DINT := 120;
	INDEX_VALIDATE_RETURNSPROPERRESULTBASEDONPERMISSIVES							: DINT := 121;
	INDEX_VALIDATE_WITHCONTINUOUSEVALUATION_PROPER									: DINT := 122;
	INDEX_VALIDATIONOK_INTERLOCKDROPDURINGEXECUTION									: DINT := 123;
	INDEX_VALIDCOMMAND_EXPECTEXECUTED_PROPER										: DINT := 124;
END_VAR

VAR

	// Mock component for testing
	MockComponent 			: FB_ComponentDerivative;

	// Common test interfaces for all methods (FB-level for stability)
	// Initialized to 0 to prevent page faults - will be set by each test method safely
	iTestCommand 			: I_CommandUnderTest;
	iTestCommandConfig 		: I_CommandConfiguration;
	iTestComponent 			: I_ComponentFull;
	iTestPermIntlkConfig 	: I_PermIntlkConfiguration;
	iTestPermIntlk 			: I_PermIntlk;
	iTestPermIntlkEval		: I_PermIntlk;
	
	// Array instances for test methods (indices 0-17)
	TestCommand : ARRAY[GC_Test.INDEX_TestFB_Command_MIN..GC_Test.INDEX_TestFB_Command_MAX] OF FB_CommandUnderTest;
	TestComponent : ARRAY[GC_Test.INDEX_TestFB_Command_MIN..GC_Test.INDEX_TestFB_Command_MAX] OF FB_ComponentDerivative;
	TestCommandConfig : ARRAY[GC_Test.INDEX_TestFB_Command_MIN..GC_Test.INDEX_TestFB_Command_MAX] OF FB_CmdPermIntlkConfiguration;
	TestPermIntlk : ARRAY[GC_Test.INDEX_TestFB_Command_MIN..GC_Test.INDEX_TestFB_Command_MAX] OF FB_PermIntlkCommand;
	MockQueue : ARRAY[GC_Test.INDEX_TestFB_Command_MIN..GC_Test.INDEX_TestFB_Command_MAX] OF FB_RingBufferICmd;
	CommandTimer : ARRAY[GC_Test.INDEX_TestFB_Command_MIN..GC_Test.INDEX_TestFB_Command_MAX] OF FB_CommandElapsedTimer;
//	FileHandler : ARRAY[GC_Test.INDEX_TestFB_Command_MIN..GC_Test.INDEX_TestFB_Command_MAX] OF FB_FileHandlerCsv;
END_VAR

// ================================================================
// ACTIVE TESTS - BehaviorTests, FaultInjectionTests, StateDrivenCompletenessTests, IntegrationTests
// ================================================================

// Tests previously listed here have been moved to a consolidated section below
TEST_Forbidden_ResumeWithoutPermissive_ReturnsForbidden();

// Priority tests - implemented
TEST_InjectConfigurations_StoresInterfacesProperly();
TEST_Validate_ReturnsProperResultBasedOnPermissives();
TEST_Validate_WithContinuousEvaluation();
TEST_ValidationOK_InterlockDropDuringExecution();
TEST_CommandTimeout_TriggersReset();
TEST_Reset_ClearsCommandState();
TEST_Execute_TransitionsFromAcceptedToOk();

// Edge-triggered functionality tests  
TEST_EdgeTriggered_StateMachineExecution();
TEST_StepState_TransitionsAndValidation(); 
TEST_CyclicLogic_StateMachineProgression();
//TEST_FileHandler_EdgeTriggeredOperations();

// TIER 1: SAFETY CRITICAL - Migrated from FB_ComponentTests
TEST_PermIntlkLostDuringBusy_CommandAbortedWithInterlockLost();
TEST_ComponentBusyDuringValidation_ResultConflict();
TEST_PermissiveFalseDuringValidation_ResultForbidden();

// TIER 2: OPERATIONAL CRITICAL - Command State Management
TEST_CommandCompletes_StatusDoneAndBusyCleared();
TEST_CommandAttemptsExceedRetryCount_ResultTooManyRequests();

// Additional command lifecycle tests
TEST_ValidCommand_ExpectExecuted();
GivenCommandAlreadyRunning_WhenExecute_ExpectConflictResult();
GivenCommand_WhenResetCalled_ExpectStateCleared();
GivenCommand_WhenValidateCalled_ExpectValidationResultMatchesConfiguration();


// Error result preservation tests
TEST_CompleteState_PreservesTimeoutResult();
TEST_CompleteState_PreservesAbortedResult();
TEST_AbortAfterComplete_StatePreservation();
TEST_CompleteState_SetsOkForSuccessfulCompletion();

// New functionality tests for identified issues
TEST_Cancel_FromQueuedState();
TEST_Execute_StateMachineProgression();

// Advanced architectural validation tests
TEST_OperatorAbort_VsInterlockAbort_DifferentResults();
TEST_PauseResume_StateTransitions();
TEST_TerminalResults_ErrorFlagConsistency();

// Configuration and state tests
GivenValidConfiguration_WhenInjectConfigurationCalled_ExpectConfigurationStored();
GivenInvalidConfiguration_WhenInjectConfigurationCalled_ExpectInitializationFailure();
GivenTimerStarted_WhenCyclicLogicRuns_ExpectElapsedTimeIncreases();
GivenCommandExecuted_WhenCyclicLogicRuns_ExpectStateProgression();

GivenCommandQueued_WhenAbort_ExpectCommandAbortedAndStatusUpdated();
GivenCommandPaused_WhenAbort_ExpectCommandAbortedAndStatusUpdated();
GivenCommandQueued_WhenCancel_ExpectCommandRemovedFromQueue();
GivenCommandPaused_WhenResume_ExpectCommandResumesExecution();
GivenRunningCommand_WhenPause_ExpectCommandTransitionsToPausedState();
GivenCommandInIdleState_WhenCancel_ExpectNoActionTaken();
GivenInjectedConfigurationsValid_WhenInjectConfigurations_ExpectInterfacesStoredAndInitialized();
GivenInvalidConfigurations_WhenInjectConfigurations_ExpectInitializationFailure();
GivenComponentReset_WhenResetCalled_ExpectAllCommandStateCleared();
GivenCommandValidated_WhenValidateCalled_ExpectTrue();
GivenCommandInvalid_WhenValidateCalled_ExpectFalse();
GivenCommand_WhenExecuteCalled_ExpectExecutionOccurs();
GivenCommand_WhenCancelCalledIfCommandNotAlreadyDequeuedExpectCommandRemovedFromQueue();
GivenCommand_WhenPauseCalledExpectCommandPauses();
GivenCommand_WhenResumeCalledExpectCommandResumes();
GivenCommand_WhenQueueCalledExpectCommandAddedToQueue();
GivenCommand_WhenValidateCalled_ExpectPermissiveOK();
TEST_InterfaceInjectionConfigurationResolution();
GivenCommand_WhenCyclicLogicCalled_ExpectStateUpdated();
GivenTimerStopped_WhenCyclicLogicRuns_ExpectElapsedTimeRemainsConstant();

// Tests from systematic state coverage section onwards moved to FB_CommandTestsII

METHOD PRIVATE GivenCommand_WhenCancelCalledIfCommandNotAlreadyDequeuedExpectCommandRemovedFromQueue
VAR
	TestIdx : DINT := INDEX_GIVENCOMMAND_WHENCANCEL_EXPECTREMOVEDFROMQUEUE;
END_VAR
TEST(__POUNAME());

// Initialize test objects first
TestCommand[TestIdx].Initialize();
TestComponent[TestIdx].Initialize();
TestCommandConfig[TestIdx].Initialize();
TestPermIntlk[TestIdx].Initialize();

// Safe interface assignments using __QUERYINTERFACE for validation
iTestCommand := TestCommand[TestIdx];

iTestCommandConfig := TestCommandConfig[TestIdx];

iTestComponent := TestComponent[TestIdx];

iTestPermIntlkConfig := TestCommandConfig[TestIdx];

// Interface validation with protection
IF iTestCommand = 0 THEN
	AssertTrue(Condition := FALSE, Message := 'TEST FAILED: iTestCommand interface is null - cannot execute test');
	RETURN;
END_IF

IF iTestCommandConfig = 0 THEN
	AssertTrue(Condition := FALSE, Message := 'TEST FAILED: iTestCommandConfig interface is null - cannot execute test');
	RETURN;
END_IF

IF iTestComponent = 0 THEN
	AssertTrue(Condition := FALSE, Message := 'TEST FAILED: iTestComponent interface is null - cannot execute test');
	RETURN;
END_IF

// Configure command
iTestCommandConfig.P_CommandConfiguration.CommandDescription := 'Test Cancel Command Not Already Dequeued';
IF __ISVALIDREF(iTestCommandConfig.P_CommandConfiguration.BaseConfiguration) THEN
    iTestCommandConfig.P_CommandConfiguration.BaseConfiguration.LogTraceConfiguration.When := E_LogTraceWhen.xRunOnInitOnly;
END_IF

// Setup command with configurations
iTestCommand.InjectConfigurations(
	iComponent := iTestComponent,
	iCommandConfiguration := iTestCommandConfig,
	iPermIntlkConfiguration := iTestPermIntlkConfig
);

// Queue the command
iTestCommand.Queue();

AssertTrue(
	Condition := iTestCommand.P_CommandStatus.StepState = E_CommandState.Idle,
	Message := 'Command should be queued before cancel'
);

AssertEquals_UDINT(
	Expected := E_CommandResult.Accepted,
	Actual := iTestCommand.P_CommandStatus.Result,
	Message := 'Queue should set Result to Accepted'
);

// Cancel the command (should remove from queue if not already dequeued)
iTestCommand.Cancel();

// Verify Cancel set Result to Cancelled and StepState to Idle per review guidance
AssertEquals_UDINT(
	Expected := E_CommandResult.Cancelled,
	Actual := iTestCommand.P_CommandStatus.Result,
	Message := 'Command result should be Cancelled after calling Cancel()'
);

AssertEquals_UDINT(
	Expected := E_CommandState.Idle,
	Actual := iTestCommand.P_CommandStatus.StepState,
	Message := 'Command should return to Idle state after Cancel'
);

TEST_FINISHED();
END_METHOD

METHOD PRIVATE GivenCommand_WhenExecuteCalled_ExpectExecutionOccurs
VAR
	TestIdx : DINT := INDEX_GIVENCOMMAND_WHENEXECUTECALLED_EXPECTEXECUTION;
END_VAR
TEST(__POUNAME());

// Initialize test objects first
TestCommand[TestIdx].Initialize();
TestComponent[TestIdx].Initialize();
TestCommandConfig[TestIdx].Initialize();
TestPermIntlk[TestIdx].Initialize();

// Safe interface assignments using __QUERYINTERFACE for validation
iTestCommand := TestCommand[TestIdx];

iTestCommandConfig := TestCommandConfig[TestIdx];

iTestComponent := TestComponent[TestIdx];

iTestPermIntlkConfig := TestCommandConfig[TestIdx];

// Interface validation with protection
IF iTestCommand = 0 THEN
	AssertTrue(Condition := FALSE, Message := 'TEST FAILED: iTestCommand interface is null - cannot execute test');
	RETURN;
END_IF

IF iTestCommandConfig = 0 THEN
	AssertTrue(Condition := FALSE, Message := 'TEST FAILED: iTestCommandConfig interface is null - cannot execute test');
	RETURN;
END_IF

IF iTestComponent = 0 THEN
	AssertTrue(Condition := FALSE, Message := 'TEST FAILED: iTestComponent interface is null - cannot execute test');
	RETURN;
END_IF

// Configure command
iTestCommandConfig.P_CommandConfiguration.CommandDescription := 'Test Command Execution';
IF __ISVALIDREF(iTestCommandConfig.P_CommandConfiguration.BaseConfiguration) THEN
    iTestCommandConfig.P_CommandConfiguration.BaseConfiguration.LogTraceConfiguration.When := E_LogTraceWhen.xRunOnInitOnly;
END_IF

// Configure permissive to be OK for successful validation
IF iTestPermIntlkConfig <> 0 THEN
	iTestPermIntlkConfig.P_PermIntlkConfiguration.PermIntlkObj[1].Description := 'Test Permissive';
	iTestPermIntlkConfig.P_PermIntlkConfiguration.PermIntlkObj[1].Condition := TRUE;
	iTestPermIntlkConfig.P_PermIntlkConfiguration.PermIntlkObj[1].Index := 1;
END_IF

// Setup command with configurations
iTestCommand.InjectConfigurations(
	iComponent := iTestComponent,
	iCommandConfiguration := iTestCommandConfig,
	iPermIntlkConfiguration := iTestPermIntlkConfig
);

// Verify command is ready for execution
AssertTrue(
	Condition := iTestCommand.P_CommandStatus.BaseStatus.Initialized,
	Message := 'Command should be initialized before execution'
);

AssertFalse(
	Condition := iTestCommand.P_CommandStatus.BaseStatus.Busy,
	Message := 'Command should not be busy before execution'
);

// First validate the command (component pattern: validate then execute)
iTestCommand.Validate();

// Verify validation succeeded
AssertEquals_UDINT(
	Expected := E_CommandResult.Accepted,
	Actual := iTestCommand.P_CommandStatus.Result,
	Message := 'Command should be Accepted after validation'
);

// Execute the command
iTestCommand.Execute();

// Verify execution occurred
AssertTrue(
	Condition := iTestCommand.P_CommandStatus.BaseStatus.Busy,
	Message := 'Command should be busy after Execute() is called'
);

AssertEquals_UDINT(
	Expected := E_CommandResult.Accepted,
	Actual := iTestCommand.P_CommandStatus.Result,
	Message := 'Command result should be Accepted after Execute() is called'
);

// Run cyclic logic to progress execution
iTestCommand.CyclicLogic();

// Verify execution is progressing
AssertTrue(
	Condition := iTestCommand.P_CommandStatus.BaseStatus.Busy OR iTestCommand.P_CommandStatus.BaseStatus.Done,
	Message := 'Command should be busy or done after cyclic logic execution'
);

TEST_FINISHED();
END_METHOD

METHOD PRIVATE GivenCommand_WhenQueueCalledExpectCommandAddedToQueue
VAR
	TestIdx : DINT := INDEX_GIVENCOMMAND_WHENQUEUECALLED_EXPECTADDEDTOQUEUE;
END_VAR
TEST(__POUNAME());

// Initialize test objects first
TestCommand[TestIdx].Initialize();
TestComponent[TestIdx].Initialize();
TestCommandConfig[TestIdx].Initialize();
TestPermIntlk[TestIdx].Initialize();

// Safe interface assignments using __QUERYINTERFACE for validation
iTestCommand := TestCommand[TestIdx];

iTestCommandConfig := TestCommandConfig[TestIdx];

iTestComponent := TestComponent[TestIdx];

iTestPermIntlkConfig := TestPermIntlk[TestIdx];

// Interface validation with protection
IF iTestCommand = 0 THEN
	AssertTrue(Condition := FALSE, Message := 'TEST FAILED: iTestCommand interface is null - cannot execute test');
	RETURN;
END_IF

IF iTestCommandConfig = 0 THEN
	AssertTrue(Condition := FALSE, Message := 'TEST FAILED: iTestCommandConfig interface is null - cannot execute test');
	RETURN;
END_IF

IF iTestComponent = 0 THEN
	AssertTrue(Condition := FALSE, Message := 'TEST FAILED: iTestComponent interface is null - cannot execute test');
	RETURN;
END_IF

// Configure command
iTestCommandConfig.P_CommandConfiguration.CommandDescription := 'Test Command Queue';
IF __ISVALIDREF(iTestCommandConfig.P_CommandConfiguration.BaseConfiguration) THEN
    iTestCommandConfig.P_CommandConfiguration.BaseConfiguration.LogTraceConfiguration.When := E_LogTraceWhen.xRunOnInitOnly;
END_IF

// Configure permissive to be OK
IF iTestPermIntlkConfig <> 0 THEN
	iTestPermIntlkConfig.P_PermIntlkConfiguration.PermIntlkObj[1].Description := 'Test Permissive';
	iTestPermIntlkConfig.P_PermIntlkConfiguration.PermIntlkObj[1].Condition := TRUE;
	iTestPermIntlkConfig.P_PermIntlkConfiguration.PermIntlkObj[1].Index := 1;
END_IF

// Setup command with configurations
iTestCommand.InjectConfigurations(
	iComponent := iTestComponent,
	iCommandConfiguration := iTestCommandConfig,
	iPermIntlkConfiguration := iTestPermIntlkConfig
);

// Resolve configurations after injection
iTestCommand.CyclicLogic();

// Verify command starts in Idle state (normal initial state)
AssertEquals_UDINT(
	Expected := E_CommandState.Idle,
	Actual := iTestCommand.P_CommandStatus.StepState,
	Message := 'Command should start in Idle state'
);

// Verify command is not yet queued (result should not be Accepted yet)
AssertTrue(
	Condition := iTestCommand.P_CommandStatus.Result <> E_CommandResult.Accepted,
	Message := 'Command should not have Accepted result before queuing'
);

// Queue the command
iTestCommand.Queue();

// Verify command was added to queue - Queued semantics also require Result==Accepted
AssertTrue(
	Condition := iTestCommand.P_CommandStatus.StepState = E_CommandState.Idle,
	Message := 'Command should be queued after calling Queue()'
);

AssertEquals_UDINT(
	Expected := E_CommandResult.Accepted,
	Actual := iTestCommand.P_CommandStatus.Result,
	Message := 'Queue should set Result to Accepted (queued commands have Accepted result)'
);

TEST_FINISHED();
END_METHOD

METHOD PRIVATE GivenCommand_WhenResetCalled_ExpectStateCleared
VAR
	TestIdx : DINT := INDEX_GIVENCOMMAND_WHENRESETCALLED_EXPECTSTATECLEARED;
END_VAR
TEST(__POUNAME());

// Initialize test objects first - Use index 101 to avoid conflicts
TestCommand[TestIdx].Initialize();
TestComponent[TestIdx].Initialize();
TestCommandConfig[TestIdx].Initialize();
TestPermIntlk[TestIdx].Initialize();

// Safe interface assignments using __QUERYINTERFACE for validation
iTestCommand := TestCommand[TestIdx];

iTestCommandConfig := TestCommandConfig[TestIdx];

iTestComponent := TestComponent[TestIdx];

iTestPermIntlkConfig := TestCommandConfig[TestIdx];


// Interface validation with protection
IF iTestCommand = 0 THEN
	AssertTrue(Condition := FALSE, Message := 'TEST FAILED: iTestCommand interface is null - cannot execute test');
	RETURN;
END_IF

IF iTestCommandConfig = 0 THEN
	AssertTrue(Condition := FALSE, Message := 'TEST FAILED: iTestCommandConfig interface is null - cannot execute test');
	RETURN;
END_IF

IF iTestComponent = 0 THEN
	AssertTrue(Condition := FALSE, Message := 'TEST FAILED: iTestComponent interface is null - cannot execute test');
	RETURN;
END_IF

// Configure command
iTestCommandConfig.P_CommandConfiguration.CommandDescription := 'Test Command Reset';
IF __ISVALIDREF(iTestCommandConfig.P_CommandConfiguration.BaseConfiguration) THEN
    iTestCommandConfig.P_CommandConfiguration.BaseConfiguration.LogTraceConfiguration.When := E_LogTraceWhen.xRunOnInitOnly;
END_IF

// Setup command with configurations
iTestCommand.InjectConfigurations(
	iComponent := iTestComponent,
	iCommandConfiguration := iTestCommandConfig,
	iPermIntlkConfiguration := iTestPermIntlkConfig
);

// Start and abort command to create some state
iTestCommand.Execute();
iTestCommand.CyclicLogic(); // Make command busy
iTestCommand.Abort(); // Create aborted state

// Verify initial state before reset
AssertEquals_UDINT(
	Expected := E_CommandResult.Aborted,
	Actual := iTestCommand.P_CommandStatus.Result,
	Message := 'Command should be Aborted before reset'
);

// Reset the command
iTestCommand.Reset();
iTestCommand.CyclicLogic(); // Process the reset

// Verify all state was cleared
AssertEquals_UDINT(
	Expected := E_CommandResult.None,
	Actual := iTestCommand.P_CommandStatus.Result,
	Message := 'Command result should be None after reset'
);

AssertEquals_UDINT(
	Expected := E_CommandState.Idle,
	Actual := iTestCommand.P_CommandStatus.StepState,
	Message := 'Command should be in Idle state after reset'
);

AssertFalse(
	Condition := iTestCommand.P_CommandStatus.BaseStatus.Busy,
	Message := 'Busy flag should be cleared after reset'
);

AssertFalse(
	Condition := iTestCommand.P_CommandStatus.BaseStatus.Done,
	Message := 'Done flag should be cleared after reset'
);

AssertFalse(
	Condition := iTestCommand.P_CommandStatus.BaseStatus.Error,
	Message := 'Error flag should be cleared after reset'
);

AssertEquals_DINT(
	Expected := 0,
	Actual := iTestCommand.P_CommandStatus.CommandTryCount,
	Message := 'CommandTryCount should be reset to 0'
);

// Verify command is ready for reuse after reset
iTestCommand.Execute();
AssertEquals_UDINT(
	Expected := E_CommandResult.Accepted,
	Actual := iTestCommand.P_CommandStatus.Result,
	Message := 'Command should be ready for reuse after reset - Execute should work'
);

TEST_FINISHED();
END_METHOD

METHOD PRIVATE GivenCommandInIdleState_WhenCancel_ExpectNoActionTaken
VAR
	TestIdx : DINT := INDEX_GIVENCOMMANDINIDLESTATE_WHENCANCEL_EXPECTNOACTIONTAKEN;
	initialResult : UDINT;
	initialBusy : BOOL;
	initialDone : BOOL;
	initialStepState : UDINT;
END_VAR
TEST(__POUNAME());

// Initialize test objects first
TestCommand[TestIdx].Initialize();
TestComponent[TestIdx].Initialize();
TestCommandConfig[TestIdx].Initialize();
TestPermIntlk[TestIdx].Initialize();

// Safe interface assignments using __QUERYINTERFACE for validation
iTestCommand := TestCommand[TestIdx];

iTestCommandConfig := TestCommandConfig[TestIdx];

iTestComponent := TestComponent[TestIdx];

iTestPermIntlkConfig := TestPermIntlk[TestIdx];


// Interface validation with protection
IF iTestCommand = 0 THEN
	AssertTrue(Condition := FALSE, Message := 'TEST FAILED: iTestCommand interface is null - cannot execute test');
	RETURN;
END_IF

IF iTestCommandConfig = 0 THEN
	AssertTrue(Condition := FALSE, Message := 'TEST FAILED: iTestCommandConfig interface is null - cannot execute test');
	RETURN;
END_IF

IF iTestComponent = 0 THEN
	AssertTrue(Condition := FALSE, Message := 'TEST FAILED: iTestComponent interface is null - cannot execute test');
	RETURN;
END_IF

// Configure command
iTestCommandConfig.P_CommandConfiguration.CommandDescription := 'Test Command Idle State Cancel';
IF __ISVALIDREF(iTestCommandConfig.P_CommandConfiguration.BaseConfiguration) THEN
    iTestCommandConfig.P_CommandConfiguration.BaseConfiguration.LogTraceConfiguration.When := E_LogTraceWhen.xRunOnInitOnly;
END_IF

// Configure permissive to be OK
IF iTestPermIntlkConfig <> 0 THEN
	iTestPermIntlkConfig.P_PermIntlkConfiguration.PermIntlkObj[1].Description := 'Test Permissive';
	iTestPermIntlkConfig.P_PermIntlkConfiguration.PermIntlkObj[1].Condition := TRUE;
	iTestPermIntlkConfig.P_PermIntlkConfiguration.PermIntlkObj[1].Index := 1;
END_IF

// Setup command with configurations
iTestCommand.InjectConfigurations(
	iComponent := iTestComponent,
	iCommandConfiguration := iTestCommandConfig,
	iPermIntlkConfiguration := iTestPermIntlkConfig
);

// Resolve configurations after injection
iTestCommand.CyclicLogic();

// Command is initialized - verify initial Idle state
AssertEquals_UDINT(
	Expected := E_CommandState.Idle,
	Actual := iTestCommand.P_CommandStatus.StepState,
	Message := 'Command should be in Idle state after initialization'
);

// Store initial state for comparison
initialResult := iTestCommand.P_CommandStatus.Result;
initialBusy := iTestCommand.P_CommandStatus.BaseStatus.Busy;
initialDone := iTestCommand.P_CommandStatus.BaseStatus.Done;
initialStepState := iTestCommand.P_CommandStatus.StepState;

// Note: Just capture initial result - don't assert a specific value since it depends on configuration state
// The important test is that Cancel() doesn't change this initial result

// Cancel the command in Idle state
iTestCommand.Cancel();

// Process the cancel operation  
iTestCommand.CyclicLogic();

// Verify no action was taken - all state should remain unchanged
AssertEquals_UDINT(
	Expected := initialResult,
	Actual := iTestCommand.P_CommandStatus.Result,
	Message := 'Command result should remain unchanged when cancelling Idle command'
);

AssertEquals_BOOL(
	Expected := initialBusy,
	Actual := iTestCommand.P_CommandStatus.BaseStatus.Busy,
	Message := 'Command busy state should remain unchanged when cancelling Idle command'
);

AssertEquals_BOOL(
	Expected := initialDone,
	Actual := iTestCommand.P_CommandStatus.BaseStatus.Done,
	Message := 'Command done state should remain unchanged when cancelling Idle command'
);

AssertEquals_UDINT(
	Expected := initialStepState,
	Actual := iTestCommand.P_CommandStatus.StepState,
	Message := 'Command step state should remain unchanged when cancelling Idle command'
);

// Verify command is still in Idle state after cancel operation
AssertEquals_UDINT(
	Expected := E_CommandState.Idle,
	Actual := iTestCommand.P_CommandStatus.StepState,
	Message := 'Command should remain in Idle state after cancel operation'
);

TEST_FINISHED();
END_METHOD

METHOD PRIVATE GivenCommandPaused_WhenAbort_ExpectCommandAbortedAndStatusUpdated
VAR
	TestIdx : DINT := INDEX_GIVENCOMMANDPAUSED_WHENABORT_EXPECTCOMMANDABORTEDANDSTATUSUPDATED;
END_VAR
TEST(__POUNAME());

// Initialize test objects first
TestCommand[TestIdx].Initialize();
TestComponent[TestIdx].Initialize();
TestCommandConfig[TestIdx].Initialize();

// Safe interface assignments using __QUERYINTERFACE for validation
iTestCommand := TestCommand[TestIdx];

iTestCommandConfig := TestCommandConfig[TestIdx];

iTestComponent := TestComponent[TestIdx];


// Interface validation with protection
IF iTestCommand = 0 THEN
	AssertTrue(Condition := FALSE, Message := 'TEST FAILED: iTestCommand interface is null - cannot execute test');
	RETURN;
END_IF

IF iTestCommandConfig = 0 THEN
	AssertTrue(Condition := FALSE, Message := 'TEST FAILED: iTestCommandConfig interface is null - cannot execute test');
	RETURN;
END_IF

IF iTestComponent = 0 THEN
	AssertTrue(Condition := FALSE, Message := 'TEST FAILED: iTestComponent interface is null - cannot execute test');
	RETURN;
END_IF

// Configure command
iTestCommandConfig.P_CommandConfiguration.CommandDescription := 'Test Paused Command Abort';
IF __ISVALIDREF(iTestCommandConfig.P_CommandConfiguration.BaseConfiguration) THEN
    iTestCommandConfig.P_CommandConfiguration.BaseConfiguration.LogTraceConfiguration.When := E_LogTraceWhen.xRunOnInitOnly;
END_IF

// Setup command with configurations
iTestCommand.InjectConfigurations(
	iComponent := iTestComponent,
	iCommandConfiguration := iTestCommandConfig,
	iPermIntlkConfiguration := iTestPermIntlkConfig
);

// Execute then pause the command
iTestCommand.Execute();
iTestCommand.CyclicLogic(); // Make command busy
iTestCommand.Pause();

AssertTrue(
	Condition := iTestCommand.P_CommandStatus.StepState = E_CommandState.Paused,
	Message := 'Command should be paused before abort'
);

// Abort the paused command
iTestCommand.Abort();

// Verify command was aborted
AssertEquals_UDINT(
	Expected := E_CommandResult.Aborted,
	Actual := iTestCommand.P_CommandStatus.Result,
	Message := 'Command result should be Aborted after calling Abort()'
);

AssertFalse(
	Condition := iTestCommand.P_CommandStatus.StepState = E_CommandState.Paused,
	Message := 'Command should not be paused after abort'
);

AssertFalse(
	Condition := iTestCommand.P_CommandStatus.BaseStatus.Busy,
	Message := 'Command should not be busy after abort from paused state'
);

TEST_FINISHED();
END_METHOD

METHOD PRIVATE GivenCommandQueued_WhenAbort_ExpectCommandAbortedAndStatusUpdated
VAR
	TestIdx : DINT := INDEX_GIVENCOMMANDQUEUED_WHENABORT_EXPECTCOMMANDABORTEDANDSTATUSUPDATED;
END_VAR
TEST(__POUNAME());

// Initialize test objects first - Use index 102 to avoid conflicts
TestCommand[TestIdx].Initialize();
TestComponent[TestIdx].Initialize();
TestCommandConfig[TestIdx].Initialize();
TestPermIntlk[TestIdx].Initialize();

// Safe interface assignments using __QUERYINTERFACE for validation
iTestCommand := TestCommand[TestIdx];

iTestCommandConfig := TestCommandConfig[TestIdx];

iTestComponent := TestComponent[TestIdx];

iTestPermIntlkConfig := TestPermIntlk[TestIdx];


// Interface validation with protection
IF iTestCommand = 0 THEN
	AssertTrue(Condition := FALSE, Message := 'TEST FAILED: iTestCommand interface is null - cannot execute test');
	RETURN;
END_IF

IF iTestCommandConfig = 0 THEN
	AssertTrue(Condition := FALSE, Message := 'TEST FAILED: iTestCommandConfig interface is null - cannot execute test');
	RETURN;
END_IF

IF iTestComponent = 0 THEN
	AssertTrue(Condition := FALSE, Message := 'TEST FAILED: iTestComponent interface is null - cannot execute test');
	RETURN;
END_IF

// Configure command
iTestCommandConfig.P_CommandConfiguration.CommandDescription := 'Test Queued Command Cancel';
IF __ISVALIDREF(iTestCommandConfig.P_CommandConfiguration.BaseConfiguration) THEN
    iTestCommandConfig.P_CommandConfiguration.BaseConfiguration.LogTraceConfiguration.When := E_LogTraceWhen.xRunOnInitOnly;
END_IF

// Configure permissive to be OK
IF iTestPermIntlkConfig <> 0 THEN
	iTestPermIntlkConfig.P_PermIntlkConfiguration.PermIntlkObj[1].Description := 'Test Permissive';
	iTestPermIntlkConfig.P_PermIntlkConfiguration.PermIntlkObj[1].Condition := TRUE;
	iTestPermIntlkConfig.P_PermIntlkConfiguration.PermIntlkObj[1].Index := 1;
END_IF

// Setup command with configurations
iTestCommand.InjectConfigurations(
	iComponent := iTestComponent,
	iCommandConfiguration := iTestCommandConfig,
	iPermIntlkConfiguration := iTestPermIntlkConfig
);

// Resolve configurations after injection
iTestCommand.CyclicLogic();

// Queue the command (keep it in Idle state - queued commands are in Idle)
iTestCommand.Queue();

AssertEquals_UDINT(
	Expected := E_CommandState.Idle,
	Actual := iTestCommand.P_CommandStatus.StepState,
	Message := 'Command should be in Idle state when queued'
);

// Cancel the queued command (queued commands can only be cancelled, not aborted)
iTestCommand.Cancel();

// Verify command was cancelled and status updated
AssertEquals_UDINT(
	Expected := E_CommandResult.Cancelled,
	Actual := iTestCommand.P_CommandStatus.Result,
	Message := 'Queued command result should be Cancelled after calling Cancel()'
);

AssertEquals_UDINT(
	Expected := E_CommandState.Idle,
	Actual := iTestCommand.P_CommandStatus.StepState,
	Message := 'Command should remain in Idle state after cancel (removed from queue)'
);

AssertFalse(
	Condition := iTestCommand.P_CommandStatus.BaseStatus.Busy,
	Message := 'Command should not be busy after cancel from queued state'
);

TEST_FINISHED();
END_METHOD

METHOD PRIVATE GivenCommandQueued_WhenCancel_ExpectCommandRemovedFromQueue
VAR
	TestIdx : DINT := INDEX_GIVENCOMMANDQUEUED_WHENCANCEL_EXPECTCOMMANDREMOVEDFROMQUEUE;
	initialResult : UDINT;
	initialBusy : BOOL;
	initialDone : BOOL;
	initialStepState : UDINT;
END_VAR
TEST(__POUNAME());

// REDESIGNED: Commands don't actually know about queues - this tests Cancel() on Idle commands
// Queue management is handled by external systems, not the command itself
// This test verifies that Cancel() safely ignores commands in inactive states

// Initialize test objects first
TestCommand[TestIdx].Initialize();
TestComponent[TestIdx].Initialize();
TestCommandConfig[TestIdx].Initialize();
TestPermIntlk[TestIdx].Initialize();

// Safe interface assignments using __QUERYINTERFACE for validation
iTestCommand := TestCommand[TestIdx];

iTestCommandConfig := TestCommandConfig[TestIdx];

iTestComponent := TestComponent[TestIdx];

iTestPermIntlkConfig := TestPermIntlk[TestIdx];

// Interface validation with protection
IF iTestCommand = 0 THEN
	AssertTrue(Condition := FALSE, Message := 'TEST FAILED: iTestCommand interface is null - cannot execute test');
	RETURN;
END_IF

IF iTestCommandConfig = 0 THEN
	AssertTrue(Condition := FALSE, Message := 'TEST FAILED: iTestCommandConfig interface is null - cannot execute test');
	RETURN;
END_IF

IF iTestComponent = 0 THEN
	AssertTrue(Condition := FALSE, Message := 'TEST FAILED: iTestComponent interface is null - cannot execute test');
	RETURN;
END_IF

// Configure command
iTestCommandConfig.P_CommandConfiguration.CommandDescription := 'Test Cancel on Idle Command (Queue-like scenarios)';
IF __ISVALIDREF(iTestCommandConfig.P_CommandConfiguration.BaseConfiguration) THEN
    iTestCommandConfig.P_CommandConfiguration.BaseConfiguration.LogTraceConfiguration.When := E_LogTraceWhen.xRunOnInitOnly;
END_IF

// Configure permissive to be OK
IF iTestPermIntlkConfig <> 0 THEN
	iTestPermIntlkConfig.P_PermIntlkConfiguration.PermIntlkObj[1].Description := 'Test Permissive';
	iTestPermIntlkConfig.P_PermIntlkConfiguration.PermIntlkObj[1].Condition := TRUE;
	iTestPermIntlkConfig.P_PermIntlkConfiguration.PermIntlkObj[1].Index := 1;
END_IF

// Setup command with configurations
iTestCommand.InjectConfigurations(
	iComponent := iTestComponent,
	iCommandConfiguration := iTestCommandConfig,
	iPermIntlkConfiguration := iTestPermIntlkConfig
);

// Resolve configurations after injection
iTestCommand.CyclicLogic();

// TEST 1: Cancel on freshly initialized command (simulates cancel before execution)
AssertEquals_UDINT(
	Expected := E_CommandState.Idle,
	Actual := iTestCommand.P_CommandStatus.StepState,
	Message := 'Command should start in Idle state'
);

// Store initial state for comparison
initialResult := iTestCommand.P_CommandStatus.Result;
initialBusy := iTestCommand.P_CommandStatus.BaseStatus.Busy;
initialDone := iTestCommand.P_CommandStatus.BaseStatus.Done;
initialStepState := iTestCommand.P_CommandStatus.StepState;

// Cancel the idle command (simulates external queue manager cancelling queued command)
iTestCommand.Cancel();

// Process the cancel operation
iTestCommand.CyclicLogic();

// Verify Cancel() is safely ignored on idle commands
AssertEquals_UDINT(
	Expected := initialResult,
	Actual := iTestCommand.P_CommandStatus.Result,
	Message := 'Cancel should have no effect on idle command result'
);

AssertEquals_BOOL(
	Expected := initialBusy,
	Actual := iTestCommand.P_CommandStatus.BaseStatus.Busy,
	Message := 'Cancel should have no effect on idle command busy state'
);

AssertEquals_BOOL(
	Expected := initialDone,
	Actual := iTestCommand.P_CommandStatus.BaseStatus.Done,
	Message := 'Cancel should have no effect on idle command done state'
);

AssertEquals_UDINT(
	Expected := initialStepState,
	Actual := iTestCommand.P_CommandStatus.StepState,
	Message := 'Cancel should have no effect on idle command step state'
);

// TEST 2: Cancel on completed command (simulates cancel after completion)
// Execute command to completion first
iTestCommand.Execute();
iTestCommand.CyclicLogic(); // Idle -> Execute
iTestCommand.CyclicLogic(); // Execute -> Monitor
iTestCommand.CyclicLogic(); // Monitor -> Complete
iTestCommand.CyclicLogic(); // First cycle in Complete (stays Complete)
iTestCommand.CyclicLogic(); // Second cycle in Complete -> Auto-reset to Idle

// Verify command is back to idle after completion
AssertEquals_UDINT(
	Expected := E_CommandState.Idle,
	Actual := iTestCommand.P_CommandStatus.StepState,
	Message := 'Command should be idle after completion cycle'
);

// Store state after completion
initialResult := iTestCommand.P_CommandStatus.Result;
initialBusy := iTestCommand.P_CommandStatus.BaseStatus.Busy;
initialDone := iTestCommand.P_CommandStatus.BaseStatus.Done;
initialStepState := iTestCommand.P_CommandStatus.StepState;

// Cancel the completed/idle command
iTestCommand.Cancel();
iTestCommand.CyclicLogic();

// Verify Cancel() is safely ignored on completed commands too
AssertEquals_UDINT(
	Expected := initialResult,
	Actual := iTestCommand.P_CommandStatus.Result,
	Message := 'Cancel should have no effect on completed command result'
);

AssertEquals_UDINT(
	Expected := initialStepState,
	Actual := iTestCommand.P_CommandStatus.StepState,
	Message := 'Cancel should have no effect on completed command step state'
);

// TEST 3: Verify command can still execute normally after ignored cancel
iTestCommand.Execute();
AssertEquals_UDINT(
	Expected := E_CommandResult.Accepted,
	Actual := iTestCommand.P_CommandStatus.Result,
	Message := 'Command should still execute normally after ignored cancel operations'
);

TEST_FINISHED();
END_METHOD

METHOD PRIVATE GivenComponentReset_WhenResetCalled_ExpectAllCommandStateCleared
VAR
	TestIdx : DINT := INDEX_GIVENCOMPONENTRESET_WHENRESETCALLED_EXPECTALLCOMMANDSTATECLEARED;
END_VAR
TEST(__POUNAME());

// Initialize test objects first
TestCommand[TestIdx].Initialize();
TestComponent[TestIdx].Initialize();
TestCommandConfig[TestIdx].Initialize();
TestPermIntlk[TestIdx].Initialize();

// Safe interface assignments using __QUERYINTERFACE for validation
iTestCommand := TestCommand[TestIdx];

iTestCommandConfig := TestCommandConfig[TestIdx];

iTestComponent := TestComponent[TestIdx];


// Interface validation with protection
IF iTestCommand = 0 THEN
	AssertTrue(Condition := FALSE, Message := 'TEST FAILED: iTestCommand interface is null - cannot execute test');
	RETURN;
END_IF

IF iTestCommandConfig = 0 THEN
	AssertTrue(Condition := FALSE, Message := 'TEST FAILED: iTestCommandConfig interface is null - cannot execute test');
	RETURN;
END_IF

IF iTestComponent = 0 THEN
	AssertTrue(Condition := FALSE, Message := 'TEST FAILED: iTestComponent interface is null - cannot execute test');
	RETURN;
END_IF

// Configure command
iTestCommandConfig.P_CommandConfiguration.CommandDescription := 'Test Command Reset';
IF __ISVALIDREF(iTestCommandConfig.P_CommandConfiguration.BaseConfiguration) THEN
    iTestCommandConfig.P_CommandConfiguration.BaseConfiguration.LogTraceConfiguration.When := E_LogTraceWhen.xRunOnInitOnly;
END_IF

// Configure permissive to be OK for successful execution (to create busy state)
iTestPermIntlkConfig := TestPermIntlk[TestIdx];
iTestPermIntlkConfig.P_PermIntlkConfiguration.PermIntlkObj[1].Description := 'Test Permissive';
iTestPermIntlkConfig.P_PermIntlkConfiguration.PermIntlkObj[1].Condition := TRUE;
iTestPermIntlkConfig.P_PermIntlkConfiguration.PermIntlkObj[1].Index := 1;

// Setup command with configurations and execute to create state
iTestCommand.InjectConfigurations(
	iComponent := iTestComponent,
	iCommandConfiguration := iTestCommandConfig,
	iPermIntlkConfiguration := iTestPermIntlkConfig
);

// Resolve configurations after injection
iTestCommand.CyclicLogic();

iTestCommand.Execute();

// Verify execute succeeded
AssertEquals_UDINT(
	Expected := E_CommandResult.Accepted,
	Actual := iTestCommand.P_CommandStatus.Result,
	Message := 'Execute should succeed to create busy state'
);

iTestCommand.CyclicLogic(); // Create busy state

// Verify command has state before reset
AssertTrue(
	Condition := iTestCommand.P_CommandStatus.BaseStatus.Busy,
	Message := 'Command should be busy before reset to verify state exists'
);

// Create an error condition to test error flag clearing
// Simulate a permissive loss to force an error state
IF iTestPermIntlkConfig <> 0 THEN
	iTestPermIntlkConfig.P_PermIntlkConfiguration.PermIntlkObj[1].Condition := FALSE;
END_IF

iTestCommand.CyclicLogic(); // Process the permissive loss

// Verify error state was created
AssertTrue(
	Condition := iTestCommand.P_CommandStatus.BaseStatus.Error,
	Message := 'Command should have error state before reset to test error clearing'
);

// Reset command which should clear all command state
iTestCommand.Reset();

// Verify all command state was cleared
AssertFalse(
	Condition := iTestCommand.P_CommandStatus.BaseStatus.Busy,
	Message := 'Command should not be busy after command reset'
);

AssertFalse(
	Condition := iTestCommand.P_CommandStatus.BaseStatus.Done,
	Message := 'Command done flag should be cleared after command reset'
);

AssertFalse(
	Condition := iTestCommand.P_CommandStatus.BaseStatus.Error,
	Message := 'Command error flag should be cleared after command reset'
);

AssertEquals_UDINT(
	Expected := E_CommandState.Idle,
	Actual := iTestCommand.P_CommandStatus.StepState,
	Message := 'Command should be in Idle state after command reset'
);

TEST_FINISHED();
END_METHOD

METHOD PRIVATE TEST_AbortAfterComplete_StatePreservation
VAR
	TestIdx : DINT := INDEX_ABORTAFTERCOMPLETE_STATEPRESERVATION;
    stCommandStatus : ST_CommandStatus;
    stBaseStatus : ST_BaseStatus;
    stCommandConfiguration : ST_CommandConfiguration;
END_VAR
TEST(__POUNAME());

// Purpose: Checks Abort does not overwrite an already completed Ok
// Protects terminal state consistency

// Initialize reference objects
stCommandStatus.BaseStatus REF= stBaseStatus;
stCommandStatus.ConfigRef REF= stCommandConfiguration;

// === TEST 1: Abort After Successful Completion Should Not Change Ok Result ===
TestCommand[TestIdx].Initialize();
TestComponent[TestIdx].Initialize();
TestCommandConfig[TestIdx].Initialize();
TestPermIntlk[TestIdx].Initialize();

// Assign interfaces
iTestCommand := TestCommand[TestIdx];
iTestCommandConfig := TestCommandConfig[TestIdx];
iTestComponent := TestComponent[TestIdx];
iTestPermIntlkConfig := TestCommandConfig[TestIdx];

// Configure for normal completion
iTestCommandConfig.P_CommandConfiguration.CommandDescription := 'Abort After Complete Test';
iTestCommandConfig.P_CommandConfiguration.TimeoutTime := T#10S;
IF __ISVALIDREF(iTestCommandConfig.P_CommandConfiguration.BaseConfiguration) THEN
    iTestCommandConfig.P_CommandConfiguration.BaseConfiguration.LogTraceConfiguration.When := E_LogTraceWhen.xRunOnInitOnly;
END_IF

// Configure permissive to be OK for successful validation and execution
IF iTestPermIntlkConfig <> 0 THEN
	iTestPermIntlkConfig.P_PermIntlkConfiguration.PermIntlkObj[1].Description := 'Test Permissive';
	iTestPermIntlkConfig.P_PermIntlkConfiguration.PermIntlkObj[1].Condition := TRUE;
	iTestPermIntlkConfig.P_PermIntlkConfiguration.PermIntlkObj[1].Index := 1;
END_IF

iTestCommand.InjectConfigurations(
    iComponent := iTestComponent,
    iCommandConfiguration := iTestCommandConfig,
    iPermIntlkConfiguration := iTestPermIntlkConfig
);

// Initialize and resolve configurations
iTestCommand.CyclicLogic();

// Execute command to successful completion
iTestCommand.Execute();
iTestCommand.CyclicLogic(); // Execute
iTestCommand.CyclicLogic(); // Monitor
iTestCommand.Complete(); // Signal completion
iTestCommand.CyclicLogic(); // Complete

// Verify successful completion
AssertEquals_UDINT(
    Expected := E_CommandState.Complete,
    Actual := iTestCommand.P_CommandStatus.StepState,
    Message := 'Command should be in Complete state'
);

AssertEquals_UDINT(
    Expected := E_CommandResult.Ok,
    Actual := iTestCommand.P_CommandStatus.Result,
    Message := 'Command should have Ok result after successful completion'
);

AssertTrue(
    Condition := iTestCommand.P_CommandStatus.BaseStatus.Done,
    Message := 'Command should have Done=TRUE after successful completion'
);

AssertFalse(
    Condition := iTestCommand.P_CommandStatus.BaseStatus.Error,
    Message := 'Successful completion should have Error=FALSE'
);

// === CRITICAL TEST: Abort after completion should NOT overwrite Ok result ===
iTestCommand.Abort();

// Verify Ok result is preserved despite abort call
AssertEquals_UDINT(
    Expected := E_CommandResult.Ok,
    Actual := iTestCommand.P_CommandStatus.Result,
    Message := 'POLICY: Abort should NOT overwrite already completed Ok result'
);

AssertEquals_UDINT(
    Expected := E_CommandState.Complete,
    Actual := iTestCommand.P_CommandStatus.StepState,
    Message := 'POLICY: Abort should NOT change Complete state when already done'
);

AssertTrue(
    Condition := iTestCommand.P_CommandStatus.BaseStatus.Done,
    Message := 'POLICY: Abort should preserve Done=TRUE for completed command'
);

AssertFalse(
    Condition := iTestCommand.P_CommandStatus.BaseStatus.Error,
    Message := 'POLICY: Abort should not set Error=TRUE for already successful completion'
);

// === TEST 2: Abort After Error Completion Should Not Change Error Result ===
TestCommand[TestIdx].Initialize();
TestComponent[TestIdx].Initialize();
TestCommandConfig[TestIdx].Initialize();
TestPermIntlk[TestIdx].Initialize();

// Assign interfaces
iTestCommand := TestCommand[TestIdx];
iTestCommandConfig := TestCommandConfig[TestIdx];
iTestComponent := TestComponent[TestIdx];
iTestPermIntlkConfig := TestCommandConfig[TestIdx];

// Configure for timeout (error completion)
iTestCommandConfig.P_CommandConfiguration.CommandDescription := 'Abort After Error Test';
iTestCommandConfig.P_CommandConfiguration.TimeoutTime := T#1MS; // Force timeout

// Configure permissive to be OK for successful validation and execution
IF iTestPermIntlkConfig <> 0 THEN
	iTestPermIntlkConfig.P_PermIntlkConfiguration.PermIntlkObj[1].Description := 'Test Permissive';
	iTestPermIntlkConfig.P_PermIntlkConfiguration.PermIntlkObj[1].Condition := TRUE;
	iTestPermIntlkConfig.P_PermIntlkConfiguration.PermIntlkObj[1].Index := 1;
END_IF

iTestCommand.InjectConfigurations(
    iComponent := iTestComponent,
    iCommandConfiguration := iTestCommandConfig,
    iPermIntlkConfiguration := iTestPermIntlkConfig
);

// Initialize and resolve configurations
iTestCommand.CyclicLogic();

// Execute and force timeout
iTestCommand.Execute();
iTestCommand.CyclicLogic(); // Execute
iTestCommand.CyclicLogic(); // Monitor
iTestCommand.CyclicLogic(); // Should timeout

// Verify timeout completion
AssertEquals_UDINT(
    Expected := E_CommandResult.RequestTimeout,
    Actual := iTestCommand.P_CommandStatus.Result,
    Message := 'Command should have RequestTimeout result after timeout'
);

AssertTrue(
    Condition := iTestCommand.P_CommandStatus.BaseStatus.Error,
    Message := 'Timeout should set Error=TRUE'
);

// Abort after error completion should not change the error result
iTestCommand.Abort();

AssertEquals_UDINT(
    Expected := E_CommandResult.RequestTimeout,
    Actual := iTestCommand.P_CommandStatus.Result,
    Message := 'POLICY: Abort should NOT overwrite RequestTimeout result'
);

AssertTrue(
    Condition := iTestCommand.P_CommandStatus.BaseStatus.Error,
    Message := 'POLICY: Abort should preserve Error=TRUE for timeout condition'
);

// === TEST 3: Abort During Active Execution Should Work Normally ===
TestCommand[TestIdx].Initialize();
TestComponent[TestIdx].Initialize();
TestCommandConfig[TestIdx].Initialize();
TestPermIntlk[TestIdx].Initialize();

// Assign interfaces
iTestCommand := TestCommand[TestIdx];
iTestCommandConfig := TestCommandConfig[TestIdx];
iTestComponent := TestComponent[TestIdx];
iTestPermIntlkConfig := TestCommandConfig[TestIdx];

// Configure for normal execution
iTestCommandConfig.P_CommandConfiguration.CommandDescription := 'Active Abort Test';
iTestCommandConfig.P_CommandConfiguration.TimeoutTime := T#10S;

// Configure permissive to be OK for successful validation and execution
IF iTestPermIntlkConfig <> 0 THEN
	iTestPermIntlkConfig.P_PermIntlkConfiguration.PermIntlkObj[1].Description := 'Test Permissive';
	iTestPermIntlkConfig.P_PermIntlkConfiguration.PermIntlkObj[1].Condition := TRUE;
	iTestPermIntlkConfig.P_PermIntlkConfiguration.PermIntlkObj[1].Index := 1;
END_IF

iTestCommand.InjectConfigurations(
    iComponent := iTestComponent,
    iCommandConfiguration := iTestCommandConfig,
    iPermIntlkConfiguration := iTestPermIntlkConfig
);

// Initialize and resolve configurations
iTestCommand.CyclicLogic();

// Execute to active state
iTestCommand.Execute();
iTestCommand.CyclicLogic(); // Execute

// Verify active execution
AssertEquals_UDINT(
    Expected := E_CommandState.Execute,
    Actual := iTestCommand.P_CommandStatus.StepState,
    Message := 'Command should be in Execute state'
);

AssertTrue(
    Condition := iTestCommand.P_CommandStatus.BaseStatus.Busy,
    Message := 'Command should be Busy during execution'
);

// Abort during active execution should work
iTestCommand.Abort();

AssertEquals_UDINT(
    Expected := E_CommandResult.Aborted,
    Actual := iTestCommand.P_CommandStatus.Result,
    Message := 'Abort during active execution should set Aborted result'
);

AssertFalse(
    Condition := iTestCommand.P_CommandStatus.BaseStatus.Busy,
    Message := 'Abort should clear Busy flag'
);

// === TEST 4: Multiple Aborts Should Not Corrupt Terminal State ===
// Calling abort multiple times on completed command should be safe

// Reset to successful completion again
TestCommand[TestIdx].Reset();
iTestCommand.Execute();
iTestCommand.CyclicLogic(); // Execute
iTestCommand.CyclicLogic(); // Monitor
iTestCommand.Complete(); // Signal completion
iTestCommand.CyclicLogic(); // Complete

// Multiple abort calls should be harmless
iTestCommand.Abort();
iTestCommand.Abort();
iTestCommand.Abort();

// Result should remain Ok
AssertEquals_UDINT(
    Expected := E_CommandResult.Ok,
    Actual := iTestCommand.P_CommandStatus.Result,
    Message := 'Multiple aborts should not corrupt completed Ok result'
);

AssertTrue(
    Condition := iTestCommand.P_CommandStatus.BaseStatus.Done,
    Message := 'Multiple aborts should preserve Done=TRUE'
);

TEST_FINISHED();
END_METHOD

METHOD PRIVATE TEST_Cancel_FromQueuedState
VAR
	TestIdx : DINT := INDEX_CANCEL_FROMQUEUEDSTATE;
END_VAR
TEST(__POUNAME());

// Setup command in Idle state
TestCommand[TestIdx].Initialize();
TestCommandConfig[TestIdx].Initialize();

TestCommand[TestIdx].InjectConfigurations(
    iComponent := 0,
    iCommandConfiguration := TestCommandConfig[TestIdx],
    iPermIntlkConfiguration := 0
);

// Ensure command is in proper Idle state for Cancel test
TestCommand[TestIdx].Reset();

// Command starts in Idle state naturally
// Call Cancel from Idle state
TestCommand[TestIdx].Cancel();

// Verify Cancel sets proper result (Cancel from Idle should set Cancelled result)
AssertEquals_UDINT(
    Expected := E_CommandResult.Cancelled,
    Actual := TestCommand[TestIdx].P_CommandStatus.Result,
    Message := 'Cancel from Idle should set Cancelled result'
);

// State should remain Idle since we never started execution
AssertEquals_UDINT(
    Expected := E_CommandState.Idle,
    Actual := TestCommand[TestIdx].P_CommandStatus.StepState,
    Message := 'Cancel from Idle should remain in Idle state'
);

TEST_FINISHED();
END_METHOD

METHOD PRIVATE TEST_Execute_StateMachineProgression
VAR
	TestIdx : DINT := INDEX_EXECUTE_STATEMACHINEPROGRESSION;
	stCommandStatus : ST_CommandStatus;
	stBaseStatus : ST_BaseStatus;
	stCommandConfiguration : ST_CommandConfiguration;
END_VAR
TEST(__POUNAME());

// Initialize test objects first
TestCommand[TestIdx].Initialize();
TestComponent[TestIdx].Initialize();
TestCommandConfig[TestIdx].Initialize();
TestPermIntlk[TestIdx].Initialize();

// Safe interface assignments using __QUERYINTERFACE for validation
iTestCommand := TestCommand[TestIdx];

iTestCommandConfig := TestCommandConfig[TestIdx];

iTestComponent := TestComponent[TestIdx];

iTestPermIntlkConfig := TestPermIntlk[TestIdx];

// Interface validation with protection
IF iTestCommand = 0 THEN
	AssertTrue(Condition := FALSE, Message := 'TEST FAILED: iTestCommand interface is null');
	RETURN;
END_IF

// Configure the command for proper execution
iTestCommandConfig.P_CommandConfiguration.CommandDescription := 'Test State Machine Progression';
IF __ISVALIDREF(iTestCommandConfig.P_CommandConfiguration.BaseConfiguration) THEN
    iTestCommandConfig.P_CommandConfiguration.BaseConfiguration.LogTraceConfiguration.When := E_LogTraceWhen.xRunOnInitOnly;
END_IF

// Setup permissive for successful execution
IF iTestPermIntlkConfig <> 0 THEN
	iTestPermIntlkConfig.P_PermIntlkConfiguration.PermIntlkObj[1].Description := 'Execute Test Permissive';
	iTestPermIntlkConfig.P_PermIntlkConfiguration.PermIntlkObj[1].Condition := TRUE;
	iTestPermIntlkConfig.P_PermIntlkConfiguration.PermIntlkObj[1].Index := 1;
END_IF

// Setup command with configurations
iTestCommand.InjectConfigurations(
	iComponent := iTestComponent,
	iCommandConfiguration := iTestCommandConfig,
	iPermIntlkConfiguration := iTestPermIntlkConfig
);

// Initialize and resolve configurations
iTestCommand.CyclicLogic();

// Verify initial idle state
AssertEquals_UDINT(
	Expected := E_CommandState.Idle,
	Actual := iTestCommand.P_CommandStatus.StepState,
	Message := 'Command should start in Idle state'
);

AssertEquals_UDINT(
	Expected := E_CommandResult.None,
	Actual := iTestCommand.P_CommandStatus.Result,
	Message := 'Initial result should be None'
);

// Execute the command
iTestCommand.Execute();

// Verify Execute() sets Accepted result and prepares for execution
AssertEquals_UDINT(
	Expected := E_CommandResult.Accepted,
	Actual := iTestCommand.P_CommandStatus.Result,
	Message := 'Execute() should set Accepted result'
);

AssertTrue(
	Condition := iTestCommand.P_CommandStatus.BaseStatus.Busy,
	Message := 'Execute() should set Busy=TRUE'
);

// First CyclicLogic: Idle → Execute
iTestCommand.CyclicLogic();

AssertEquals_UDINT(
	Expected := E_CommandState.Execute,
	Actual := iTestCommand.P_CommandStatus.StepState,
	Message := 'First CyclicLogic should transition to Execute state'
);

AssertEquals_UDINT(
	Expected := E_CommandResult.Accepted,
	Actual := iTestCommand.P_CommandStatus.Result,
	Message := 'Result should remain Accepted during Execute state'
);

AssertTrue(
	Condition := iTestCommand.P_CommandStatus.BaseStatus.Busy,
	Message := 'Command should remain Busy during Execute state'
);

// Second CyclicLogic: Execute → Monitor
iTestCommand.CyclicLogic();

AssertEquals_UDINT(
	Expected := E_CommandState.Monitor,
	Actual := iTestCommand.P_CommandStatus.StepState,
	Message := 'Second CyclicLogic should transition to Monitor state'
);

AssertEquals_UDINT(
	Expected := E_CommandResult.Accepted,
	Actual := iTestCommand.P_CommandStatus.Result,
	Message := 'Result should remain Accepted during Monitor state'
);

AssertTrue(
	Condition := iTestCommand.P_CommandStatus.BaseStatus.Busy,
	Message := 'Command should remain Busy during Monitor state'
);

// Signal completion
iTestCommand.Complete();

// Third CyclicLogic: Monitor → Complete
iTestCommand.CyclicLogic();

AssertEquals_UDINT(
	Expected := E_CommandState.Complete,
	Actual := iTestCommand.P_CommandStatus.StepState,
	Message := 'Third CyclicLogic should transition to Complete state'
);

AssertEquals_UDINT(
	Expected := E_CommandResult.Ok,
	Actual := iTestCommand.P_CommandStatus.Result,
	Message := 'Complete state should set Ok result (converted from Accepted)'
);

AssertTrue(
	Condition := iTestCommand.P_CommandStatus.BaseStatus.Done,
	Message := 'Complete state should set Done=TRUE'
);

AssertFalse(
	Condition := iTestCommand.P_CommandStatus.BaseStatus.Busy,
	Message := 'Complete state should set Busy=FALSE'
);

TEST_FINISHED();
END_METHOD

METHOD PRIVATE TEST_Execute_TransitionsFromAcceptedToOk
VAR
	TestIdx : DINT := INDEX_EXECUTE_TRANSITIONSFROMACCEPTEDTOOK;
    stCommandStatus : ST_CommandStatus;
    stBaseStatus : ST_BaseStatus;
    stCommandConfiguration : ST_CommandConfiguration;
END_VAR
TEST(__POUNAME());

// Purpose: Validates the complete lifecycle Idle → Execute → Monitor → Complete → Ok
// This is the backbone of the command state machine

// Initialize reference objects
stCommandStatus.BaseStatus REF= stBaseStatus;
stCommandStatus.ConfigRef REF= stCommandConfiguration;

// Initialize test objects
TestCommand[TestIdx].Initialize();
TestComponent[TestIdx].Initialize();
TestCommandConfig[TestIdx].Initialize();
TestPermIntlk[TestIdx].Initialize();

// Assign interfaces
iTestCommand := TestCommand[TestIdx];
iTestCommandConfig := TestCommandConfig[TestIdx];
iTestComponent := TestComponent[TestIdx];
iTestPermIntlkConfig := TestCommandConfig[TestIdx];





// Configure command with valid timeout and permissive settings
iTestCommandConfig.P_CommandConfiguration.CommandDescription := 'Core Lifecycle Test';
iTestCommandConfig.P_CommandConfiguration.TimeoutTime := T#10S;
iTestCommandConfig.P_CommandConfiguration.AbortOnInterlockDrop := FALSE;
IF __ISVALIDREF(iTestCommandConfig.P_CommandConfiguration.BaseConfiguration) THEN
    iTestCommandConfig.P_CommandConfiguration.BaseConfiguration.LogTraceConfiguration.When := E_LogTraceWhen.xRunOnInitOnly;
END_IF

// Configure permissive to be OK for successful validation and execution
IF iTestPermIntlkConfig <> 0 THEN
	iTestPermIntlkConfig.P_PermIntlkConfiguration.PermIntlkObj[1].Description := 'Core Lifecycle Test Permissive';
	iTestPermIntlkConfig.P_PermIntlkConfiguration.PermIntlkObj[1].Condition := TRUE;
	iTestPermIntlkConfig.P_PermIntlkConfiguration.PermIntlkObj[1].Index := 1;
END_IF

// Inject configurations - this is critical for proper state machine operation
iTestCommand.InjectConfigurations(
    iComponent := iTestComponent,
    iCommandConfiguration := iTestCommandConfig,
    iPermIntlkConfiguration := iTestPermIntlkConfig
);

// Initialize and resolve configurations
iTestCommand.CyclicLogic();

// === STEP 1: Initial Idle State ===
AssertEquals_UDINT(
    Expected := E_CommandState.Idle,
    Actual := iTestCommand.P_CommandStatus.StepState,
    Message := 'Initial state should be Idle'
);

AssertEquals_UDINT(
    Expected := E_CommandResult.None,
    Actual := iTestCommand.P_CommandStatus.Result,
    Message := 'Initial result should be None'
);

AssertFalse(
    Condition := iTestCommand.P_CommandStatus.BaseStatus.Busy,
    Message := 'Initial Busy should be FALSE'
);

// === STEP 2: Execute() Sets Up Execution ===
iTestCommand.Execute();

// Execute should validate and set Accepted result immediately
AssertEquals_UDINT(
    Expected := E_CommandResult.Accepted,
    Actual := iTestCommand.P_CommandStatus.Result,
    Message := 'Execute() should set Result=Accepted immediately after validation'
);

// State should remain Idle until CyclicLogic drives progression
AssertEquals_UDINT(
    Expected := E_CommandState.Idle,
    Actual := iTestCommand.P_CommandStatus.StepState,
    Message := 'Execute() should leave StepState=Idle until CyclicLogic'
);

// Busy flag enables state transitions
AssertTrue(
    Condition := iTestCommand.P_CommandStatus.BaseStatus.Busy,
    Message := 'Execute() should set Busy=TRUE to enable transitions'
);

// Try count should be 0 until actual execution starts
AssertEquals_DINT(
    Expected := 0,
    Actual := iTestCommand.P_CommandStatus.CommandTryCount,
    Message := 'Try count should remain 0 until state progression begins'
);

// === STEP 3: First CyclicLogic → Execute State ===
iTestCommand.CyclicLogic();

AssertEquals_UDINT(
    Expected := E_CommandState.Execute,
    Actual := iTestCommand.P_CommandStatus.StepState,
    Message := 'First CyclicLogic should transition Idle → Execute'
);

AssertEquals_UDINT(
    Expected := E_CommandResult.Accepted,
    Actual := iTestCommand.P_CommandStatus.Result,
    Message := 'Result should remain Accepted during Execute state'
);

// Try count increments on first execution transition per Policy H
AssertEquals_DINT(
    Expected := 1,
    Actual := iTestCommand.P_CommandStatus.CommandTryCount,
    Message := 'Try count should increment on first transition to Execute'
);

AssertTrue(
    Condition := iTestCommand.P_CommandStatus.BaseStatus.Busy,
    Message := 'Command should remain Busy in Execute state'
);

// === STEP 4: Second CyclicLogic → Monitor State ===
iTestCommand.CyclicLogic();

AssertEquals_UDINT(
    Expected := E_CommandState.Monitor,
    Actual := iTestCommand.P_CommandStatus.StepState,
    Message := 'Second CyclicLogic should transition Execute → Monitor'
);

AssertEquals_UDINT(
    Expected := E_CommandResult.Accepted,
    Actual := iTestCommand.P_CommandStatus.Result,
    Message := 'Result should remain Accepted during Monitor state'
);

AssertTrue(
    Condition := iTestCommand.P_CommandStatus.BaseStatus.Busy,
    Message := 'Command should remain Busy in Monitor state'
);

// Signal completion
iTestCommand.Complete();

// === STEP 5: Third CyclicLogic → Complete State ===
iTestCommand.CyclicLogic();

AssertEquals_UDINT(
    Expected := E_CommandState.Complete,
    Actual := iTestCommand.P_CommandStatus.StepState,
    Message := 'Third CyclicLogic should transition Monitor → Complete'
);

// Complete state sets final result and status flags
AssertEquals_UDINT(
    Expected := E_CommandResult.Ok,
    Actual := iTestCommand.P_CommandStatus.Result,
    Message := 'Complete state should convert Accepted → Ok for success'
);

AssertTrue(
    Condition := iTestCommand.P_CommandStatus.BaseStatus.Done,
    Message := 'Complete state should set Done=TRUE'
);

AssertFalse(
    Condition := iTestCommand.P_CommandStatus.BaseStatus.Busy,
    Message := 'Complete state should set Busy=FALSE'
);

AssertFalse(
    Condition := iTestCommand.P_CommandStatus.BaseStatus.Error,
    Message := 'Successful completion should have Error=FALSE'
);

// === STEP 6: Auto-Reset After Two Cycles (Policy B) ===
// First cycle in Complete state - should remain in Complete
iTestCommand.CyclicLogic();

// Should still be in Complete state (auto-reset requires 2 cycles)
AssertEquals_UDINT(
    Expected := E_CommandState.Complete,
    Actual := iTestCommand.P_CommandStatus.StepState,
    Message := 'Command should remain in Complete state for observation (cycle 1)'
);

// Second cycle - should trigger auto-reset
iTestCommand.CyclicLogic();

// Command should auto-reset to Idle on successful completion
AssertEquals_UDINT(
    Expected := E_CommandState.Idle,
    Actual := iTestCommand.P_CommandStatus.StepState,
    Message := 'Auto-reset should return command to Idle after successful completion'
);

AssertEquals_UDINT(
    Expected := E_CommandResult.None,
    Actual := iTestCommand.P_CommandStatus.Result,
    Message := 'Auto-reset should clear Result to None'
);

AssertFalse(
    Condition := iTestCommand.P_CommandStatus.BaseStatus.Done,
    Message := 'Auto-reset should clear Done flag'
);

TEST_FINISHED();
END_METHOD

METHOD PRIVATE TEST_Reset_ClearsCommandState
VAR
	TestIdx : DINT := INDEX_RESET_CLEARSCOMMANDSTATE;
	stCommandStatus : ST_CommandStatus;
	stBaseStatus : ST_BaseStatus;
	stCommandConfiguration : ST_CommandConfiguration;
END_VAR
TEST(__POUNAME());

// Direct interface assignments
iTestCommand := TestCommand[TestIdx];
iTestCommandConfig := TestCommandConfig[TestIdx];
iTestComponent := TestComponent[TestIdx];

// Configure the command  
TestCommandConfig[TestIdx].P_CommandConfiguration.CommandDescription := 'Test Reset Clears State';

// Set up command with non-default state that needs to be cleared
stBaseStatus.Busy := TRUE;
stBaseStatus.Done := TRUE;
stBaseStatus.Error := TRUE;
stBaseStatus.ErrorID := 12345;
stCommandStatus.BaseStatus REF= stBaseStatus;
IF iTestCommandConfig <> 0 THEN
	stCommandConfiguration := iTestCommandConfig.P_CommandConfiguration;
END_IF
stCommandStatus.StepState := E_CommandState.Execute;
stCommandStatus.Result := E_CommandResult.RequestTimeout;
stCommandStatus.CommandTryCount := 3;
// Note: StartTime and ElapsedTime removed from ST_CommandStatus structure

// Inject the dirty state
iTestCommand.SetCommandStatus(stCommandStatus);

// Verify state is dirty before reset
AssertTrue(
	Condition := iTestCommand.P_CommandStatus.BaseStatus.Busy,
	Message := 'Busy should be TRUE before reset'
);

AssertEquals_UDINT(
	Expected := E_CommandResult.RequestTimeout,
	Actual := iTestCommand.P_CommandStatus.Result,
	Message := 'Result should be Timeout before reset'
);

AssertEquals_DINT(
	Expected := 3,
	Actual := iTestCommand.P_CommandStatus.CommandTryCount,
	Message := 'CommandTryCount should be 3 before reset'
);

// Call Reset method
iTestCommand.Reset();

// Verify all state was cleared
AssertFalse(
	Condition := iTestCommand.P_CommandStatus.BaseStatus.Busy,
	Message := 'Busy should be cleared after reset'
);

AssertFalse(
	Condition := iTestCommand.P_CommandStatus.BaseStatus.Done,
	Message := 'Done should be cleared after reset'
);

AssertFalse(
	Condition := iTestCommand.P_CommandStatus.BaseStatus.Error,
	Message := 'Error should be cleared after reset'
);

AssertEquals_UDINT(
	Expected := 0,
	Actual := iTestCommand.P_CommandStatus.BaseStatus.ErrorID,
	Message := 'ErrorID should be reset to 0'
);

AssertEquals_UDINT(
	Expected := E_CommandResult.None,
	Actual := iTestCommand.P_CommandStatus.Result,
	Message := 'Result should be reset to None'
);

AssertEquals_DINT(
	Expected := 0,
	Actual := iTestCommand.P_CommandStatus.CommandTryCount,
	Message := 'CommandTryCount should be reset to 0'
);

AssertEquals_UDINT(
	Expected := E_CommandState.Idle,
	Actual := iTestCommand.P_CommandStatus.StepState,
	Message := 'StepState should be reset to Idle'
);

AssertEquals_LTIME(
	Expected := LTIME#0s,
	Actual := iTestCommand.P_CommandStatus.LastCommandElapsedTime,
	Message := 'LastCommandElapsedTime should be reset to 0'
);

// Test idempotent behavior - reset again should not cause issues
iTestCommand.Reset();

AssertEquals_UDINT(
	Expected := E_CommandResult.None,
	Actual := iTestCommand.P_CommandStatus.Result,
	Message := 'Multiple resets should maintain cleared state'
);

AssertEquals_UDINT(
	Expected := E_CommandState.Idle,
	Actual := iTestCommand.P_CommandStatus.StepState,
	Message := 'Multiple resets should maintain Idle state'
);

TEST_FINISHED();
END_METHOD

METHOD PRIVATE TEST_CommandAttemptsExceedRetryCount_ResultTooManyRequests
VAR
	TestIdx : DINT := INDEX_COMMANDATTEMPTSEXCEEDRETRYCOUNT;
    stCommandStatus : ST_CommandStatus;
    stBaseStatus : ST_BaseStatus;
    stCommandConfiguration : ST_CommandConfiguration;
    retryAttempt : INT;
END_VAR
TEST(__POUNAME());

// Purpose: Validates RetryCount enforcement
// Prevents runaway retries, enforces TooManyRequests result policy

// Initialize reference objects
stCommandStatus.BaseStatus REF= stBaseStatus;
stCommandStatus.ConfigRef REF= stCommandConfiguration;

// === TEST 1: RetryCount Enforcement During Execution ===
TestCommand[TestIdx].Initialize();
TestComponent[TestIdx].Initialize();
TestCommandConfig[TestIdx].Initialize();
TestPermIntlk[TestIdx].Initialize();

// Assign interfaces
iTestCommand := TestCommand[TestIdx];
iTestCommandConfig := TestCommandConfig[TestIdx];
iTestComponent := TestComponent[TestIdx];
iTestPermIntlkConfig := TestCommandConfig[TestIdx];

// Configure with low retry limit to test enforcement
iTestCommandConfig.P_CommandConfiguration.CommandDescription := 'Retry Count Test';
iTestCommandConfig.P_CommandConfiguration.RetryCountONLYFORCOMMSENDS := 2; // Allow 2 total attempts
iTestCommandConfig.P_CommandConfiguration.TimeoutTime := T#10S;
IF __ISVALIDREF(iTestCommandConfig.P_CommandConfiguration.BaseConfiguration) THEN
    iTestCommandConfig.P_CommandConfiguration.BaseConfiguration.LogTraceConfiguration.When := E_LogTraceWhen.xRunOnInitOnly;
END_IF

// Configure permissive to be OK for successful validation and execution
IF iTestPermIntlkConfig <> 0 THEN
	iTestPermIntlkConfig.P_PermIntlkConfiguration.PermIntlkObj[1].Description := 'Retry Test Permissive';
	iTestPermIntlkConfig.P_PermIntlkConfiguration.PermIntlkObj[1].Condition := TRUE;
	iTestPermIntlkConfig.P_PermIntlkConfiguration.PermIntlkObj[1].Index := 1;
END_IF

iTestCommand.InjectConfigurations(
    iComponent := iTestComponent,
    iCommandConfiguration := iTestCommandConfig,
    iPermIntlkConfiguration := iTestPermIntlkConfig
);

// Initialize and resolve configurations
iTestCommand.CyclicLogic();

// === ATTEMPT 1: Should Succeed ===
iTestCommand.Execute();
iTestCommand.CyclicLogic(); // Transition Idle → Execute, increment TryCount

AssertEquals_UDINT(
    Expected := E_CommandResult.Accepted,
    Actual := iTestCommand.P_CommandStatus.Result,
    Message := 'First execution attempt should be accepted'
);

AssertEquals_DINT(
    Expected := 1,
    Actual := iTestCommand.P_CommandStatus.CommandTryCount,
    Message := 'Try count should be 1 on first attempt'
);

// Let this attempt fail by aborting it
iTestCommand.Abort();

